PROPERTY PUBLIC StopRequested : BOOL
GET
StopRequested := CycleStopReq;
END_GET
SET // PUBLIC
CycleStopReq := StopRequested;
END_SET
END_PROPERTY

END_FUNCTION_BLOCK

// ---- POUs/PrimeMover.TcPOU
FUNCTION_BLOCK PUBLIC PrimeMover
VAR_IN_OUT
	
END_VAR
VAR_INPUT
END_VAR
VAR_OUTPUT
END_VAR
VAR
	bInitialize : BOOL := TRUE;
	State			:	ePrimeMoverState; 
	NextState		:	ePrimeMoverState;	
	ResetCmdStatus 	:	eMM_ResetCmdStatus;
	StartupCmdStatus:	eMM_StartupCmdStatus;
	HLCStatus		:	eMM_HLCStatus;
	
	// CycleControl will send a Trigger
	Trigger: BOOL := FALSE;
	// Temporary loop variable
	COUNTER: UINT := 1;
	VehicleInitMoveTimer : TON;
	bAllVehStopped :BOOL := TRUE;
	StateTimer :TON;
	WaitAfterESTOPTimer : TON;
	SuspendAfterESTOPTimer: TON;
	bFirst : BOOL := TRUE;
END_VAR

IF (bInitialize) THEN
	bInitialize := FALSE;
	// to add all initialization code here
END_IF


CASE State OF

ePrimeMoverState.eMMUnknown:
    Status.PrimeMoverStatusMsg := 'MM: Unknown, Press Start';
	GVL_IO.MM_YEnableMagneMotion := FALSE;
    IF (GVL_IO.MC_XStartPB AND GVL_IO.MC_XAirPressureOK AND GVL_IO.MC_NotEStopped) THEN // wait for start button when powered up or PLC program restarted
		NextState := ePrimeMoverState.eMMConnect;	   
	END_IF

	StateTimer(IN:=TRUE, PT:= T#9.3S); // give a message out every 10 seconds
	IF (StateTimer.Q) THEN
		Logging.fbEventMsg.SendEventMsg(MsgClass := TCEVENTCLASS_STATEINFO, EventID:= Logging.ID_MM_Unknown, SourceID:= Logging.SrcMMPOU);
		StateTimer(IN:=FALSE);
	END_IF


ePrimeMoverState.eMMConnect:
Status.PrimeMoverStatusMsg := 'MM: Socket Connecting';	
IF (Stations.fbMMClient.eState = eSOCKET_CONNECTED) THEN
		Stations.fbMMSendMsg.M_CmdHLCStatus();
		NextState := ePrimeMoverState.eMMCheckStatus;
	END_IF

ePrimeMoverState.eMMCheckStatus:
Status.PrimeMoverStatusMsg := 'MM: Checking HLC Status';
	IF (HLCStatus = eMM_HLCStatus.eHLC_STATE_OPERATIONAL) THEN
		NextState := ePrimeMoverState.eMMSendResetCmd;		
	END_IF	

ePrimeMoverState.eMMSendResetCmd:
Status.PrimeMoverStatusMsg := 'MM: Reseting Path';
	Stations.fbMMSendMsg.M_CmdResetPath();
	ResetCmdStatus := eMM_ResetCmdStatus.eMM_ResetCmdSent;
	NextState := ePrimeMoverState.eMMWaitAccceptResetCmd;

ePrimeMoverState.eMMWaitAccceptResetCmd:
Status.PrimeMoverStatusMsg := 'MM: Waiting Reset Path ACK';
	IF (ResetCmdStatus = eMM_ResetCmdStatus.eMM_ResetCmdAck) THEN
		NextState := ePrimeMoverState.eMMWaitCmplResetCmd;			
	END_IF	

ePrimeMoverState.eMMWaitCmplResetCmd:
Status.PrimeMoverStatusMsg := 'MM: Waiting Reset Cmpl';
IF (ResetCmdStatus = eMM_ResetCmdStatus.eMM_ResetCmdComplete) THEN
		NextState := ePrimeMoverState.eMMSendStartupCmd;			
	END_IF

ePrimeMoverState.eMMSendStartupCmd:
Status.PrimeMoverStatusMsg := 'MM: Starting Up Path';
	Stations.fbMMSendMsg.M_CmdStartupPath();
	StartupCmdStatus := eMM_StartupCmdStatus.eMM_StartupCmdSent;
	NextState := ePrimeMoverState.eMMWaitAcceptStartupCmd;	

ePrimeMoverState.eMMWaitAcceptStartupCmd:
Status.PrimeMoverStatusMsg := 'MM: Waiting Startup ACK';
	IF (StartupCmdStatus = eMM_StartupCmdStatus.eMM_StartupCmdAck) THEN
		NextState := ePrimeMoverState.eMMWaitCmplStartupCmd;			
	END_IF		

ePrimeMoverState.eMMWaitCmplStartupCmd:
Status.PrimeMoverStatusMsg := 'MM: Waiting Startup CMPL';
	IF (StartupCmdStatus = eMM_StartupCmdStatus.eMM_StartupCmdComplete) THEN
		NextState := ePrimeMoverState.eMMWaitCycleControlTrigger;
	END_IF
	
ePrimeMoverState.eMMWaitCycleControlTrigger:
Status.PrimeMoverStatusMsg := 'MM: Waiting Till Safe to Index';
	IF (Trigger) THEN              //Trigger is Sent By Cycle Controller
			//NextState := ePrimeMoverState.eMMSendAllVehiclesToInitPosCmd;     
		GVL_IO.MM_YEnableMagneMotion := TRUE;
		NextState := ePrimeMoverState.eMMReadyAutoRun;     
        Trigger := FALSE;      	
	END_IF

ePrimeMoverState.eMMSendAllVehiclesToInitPosCmd:
   Trigger := FALSE;	
   FOR COUNTER := 1 TO MM_CONST.MAX_VEHICLES BY 1 DO
		Stations.fbMMSendMsg.M_CmdVehToPos(VehicleID:= COUNTER, Flags :=1, Pos := MM_CONST.GOOD_UNLOAD_POS -((COUNTER-1)* (MM_CONST.Vehicle_Length+MM_CONST.MinGapInterVehStationary)/1000), Acc := 2.0, Vel := 2.0);
		NextState := ePrimeMoverState.eMMWaitCmplAllVehiclesAtInitPos;
	END_FOR
		
ePrimeMoverState.eMMWaitCmplAllVehiclesAtInitPos:
	VehicleInitMoveTimer(IN:=TRUE,PT:=T#3S);
	IF (VehicleInitMoveTimer.Q) THEN
		bAllVehStopped := TRUE;			
		FOR COUNTER := 1 TO MM_CONST.MAX_VEHICLES BY 1 DO
			Stations.fbVehicleManager[COUNTER].VehIdle := TRUE;	
			IF (STATUS.MMVehiclesStatus[COUNTER].Velocity > 0.1) THEN //maybe get vehicle stopped by reading flags instead
				  bAllVehStopped :=FALSE;
				  Stations.fbVehicleManager[COUNTER].VehIdle := FALSE; // this additional variable helps for debug
			END_IF
		END_FOR
		IF (bAllVehStopped) THEN
			NextState := ePrimeMoverState.eMMReadyAutoRun;
			VehicleInitMoveTimer(IN:=FALSE);
		END_IF	
	END_IF 

ePrimeMoverState.eMMReadyAutoRun:
//to do handle all exceptions here 
// according to pg. 53 of 210 of MM TCP/IP manual
// When Host Controller wants to issue E-STOP, then first let all the motion come to a stop
// Then issue a Suspend Movement
// Then remove bus power

//To recover from E-STOP
// Enable Bus Power, wait
// Then issue Resume Movement...
Status.PrimeMoverStatusMsg := 'MM: Auto Run';
	IF (GVL_IO.MachineEStopped OR NOT GVL_IO.MC_XAirPressureOK) THEN 
	   SuspendAfterESTOPTimer(IN:=TRUE, PT:= T#2.5S);
	   IF (SuspendAfterESTOPTimer.Q) THEN
		   NextState := ePrimeMoverState.eMMSuspendMovement;
		   SuspendAfterESTOPTimer(IN:=FALSE);
       END_IF		
	ELSE
		SuspendAfterESTOPTimer(IN:=FALSE);
	END_IF

IF (Stations.fbMMMonitor.IsMMJammed) THEN 
	Status.PrimeMoverStatusMsg := 'MM: Jammed';
END_IF

ePrimeMoverState.eMMSuspendMovement:
	IF (bFirst) THEN 
		//Stations.fbMMSendMsg.M_CmdSuspendMov();  //Suspend command is causing more problems as it rejects commands from vehicles for movement
	END_IF
	SuspendAfterESTOPTimer(IN:=TRUE,PT:=T#5S);
	IF (SuspendAfterESTOPTimer.Q) THEN
		NextState := ePrimeMoverState.eMMESTOP;		
		SuspendAfterESTOPTimer(IN:=FALSE);
		WaitAfterESTOPTimer(IN:=FALSE);
	END_IF

ePrimeMoverState.eMMESTOP:
Status.PrimeMoverStatusMsg := 'MM: E-STOPPED';
	GVL_IO.MM_YEnableMagneMotion := FALSE;
   IF (Stations.fbCycleControl.AllowPrimeMoverEnable) THEN // wait for cycle control to tell us we are ready to move
		WaitAfterESTOPTimer(IN:=TRUE, PT:=T#5S);
		GVL_IO.MM_YEnableMagneMotion := TRUE; // Enable Magnemotion D.C. Bus and let all the vehicles move
		IF (WaitAfterESTOPTimer.Q) THEN
			//Stations.fbMMSendMsg.M_CmdResumeMov(); // let all the vehicles move
			WaitAfterESTOPTimer(IN:=FALSE);
			NextState := ePrimeMoverState.eMMReadyAutoRun;
		END_IF
       	   
	END_IF

ePrimeMoverState.eMMResumeMovement:

ePrimeMoverState.eMMError:
// to do handle all exceptions here

END_CASE

IF (State <> NextState) THEN
	bFirst := TRUE;
	StateTimer(IN:=FALSE);
ELSE
	bFirst := FALSE;
END_IF

State := NextState;

AssignStationStatusForHMI();

PROPERTY PUBLIC StartupCmdState : eMM_StartupCmdStatus
SET
StartupCmdStatus := StartupCmdState;
END_SET
END_PROPERTY

PROPERTY PUBLIC WaitingForHomingTrigger : BOOL
GET
WaitingForHomingTrigger := (StartupCmdStatus = eMM_StartupCmdStatus.eMM_StartupCmdComplete) AND (State = ePrimeMoverState.eMMWaitCycleControlTrigger);
END_GET
END_PROPERTY

METHOD PUBLIC ResetPrimeMoverAndPurge : BOOL
VAR_INPUT
END_VAR
State := ePrimeMoverState.eMMUnknown;
NextState := ePrimeMoverState.eMMUnknown;
END_METHOD

PROPERTY PUBLIC ResetCmdState : eMM_ResetCmdStatus
SET
ResetCmdStatus := ResetCmdState;
END_SET
END_PROPERTY

METHOD PUBLIC AssignStationStatusForHMI : BOOL
VAR_INPUT
END_VAR
Status.StationsState[MM_CONST.PRIME_MOVER_HMI_STATE] := State;
CASE State OF 
	ePrimeMoverState.eMMUnknown,ePrimeMoverState.eMMError:
	Status.StationStauts[MM_CONST.PRIME_MOVER_HMI_STATE] := OverallStationStatus.eError;
	
    ePrimeMoverState.eMMConnect,
	ePrimeMoverState.eMMCheckStatus,
	ePrimeMoverState.eMMSendResetCmd,
	ePrimeMoverState.eMMWaitAccceptResetCmd,
	ePrimeMoverState.eMMWaitCmplResetCmd,
	ePrimeMoverState.eMMSendStartupCmd,
	ePrimeMoverState.eMMWaitAcceptStartupCmd,
	ePrimeMoverState.eMMWaitCmplStartupCmd:
		Status.StationStauts[MM_CONST.PRIME_MOVER_HMI_STATE] := OverallStationStatus.eHoming;
	
	ePrimeMoverState.eMMWaitCycleControlTrigger:
        Status.StationStauts[MM_CONST.PRIME_MOVER_HMI_STATE] := OverallStationStatus.eWarning;
		
	ePrimeMoverState.eMMSendAllVehiclesToInitPosCmd,
	ePrimeMoverState.eMMWaitCmplAllVehiclesAtInitPos,	
    ePrimeMoverState.eMMReadyAutoRun:
	    IF (Stations.fbCycleControl.AllowPrimeMoverEnable) THEN
        	Status.StationStauts[MM_CONST.PRIME_MOVER_HMI_STATE] := OverallStationStatus.eRunning;
		ELSE 
			Status.StationStauts[MM_CONST.PRIME_MOVER_HMI_STATE] := OverallStationStatus.eCycleStop;
		END_IF
		
		IF (Stations.fbMMMonitor.IsMMJammed) THEN 
	        Status.StationStauts[MM_CONST.PRIME_MOVER_HMI_STATE] := OverallStationStatus.eError;
        END_IF
	    
		
	ELSE;	
END_CASE
END_METHOD

PROPERTY PUBLIC HLCState : eMM_HLCStatus
SET
HLCStatus := HLCState;
END_SET
END_PROPERTY

PROPERTY PUBLIC Ready : BOOL
GET
Ready := (State = ePrimeMoverState.eMMReadyAutoRun);
END_GET
END_PROPERTY

PROPERTY PUBLIC TriggerAction : BOOL
SET
Trigger := TriggerAction;
END_SET
END_PROPERTY

END_FUNCTION_BLOCK

// ---- POUs/StationManager.TcPOU
FUNCTION_BLOCK PUBLIC StationManager
VAR_INPUT
END_VAR
VAR_OUTPUT
END_VAR
VAR
END_VAR

;

METHOD PUBLIC NotifyStationNewVehArrival : BOOL
VAR_INPUT
	Pos 			:	REAL;
	StationIndex 	:	BYTE;
	VehicleID		:	BYTE;
END_VAR
CASE StationIndex OF

 
MM_CONST.LOAD_1_STA:
	Stations.fbLoad1Sta.VehicleUnderTest := VehicleID;	
    Stations.fbLoad1Sta.Trigger := TRUE;
		

MM_CONST.LOAD_2_STA:
	Stations.fbLoad2Sta.VehicleUnderTest := VehicleID;		   
    Stations.fbLoad2Sta.Trigger := TRUE;
        			
MM_CONST.LOAD_3_STA:
	Stations.fbLoad3Sta.VehicleUnderTest := VehicleID;	
	Stations.fbLoad3Sta.Trigger := TRUE;					

MM_CONST.LOAD_4_STA:					
	Stations.fbLoad4Sta.VehicleUnderTest := VehicleID;
	Stations.fbLoad4Sta.Trigger := TRUE;	

MM_CONST.STOP_BEFORE_VISION_STA:
	Stations.fbOB_StopBeforeVisionSta.VehicleUnderTest := VehicleID;
	Stations.fbOB_StopBeforeVisionSta.Trigger := TRUE;

MM_CONST.VISION_STA:
	Stations.fbVisionSta.VehicleUnderTest := VehicleID;
	Stations.fbVisionSta.Trigger := TRUE;

MM_CONST.PISTON_STA:
	Stations.fbPistonSta.VehicleUnderTest := VehicleID;
	Stations.fbPistonSta.Trigger := TRUE;

MM_CONST.CAP_STA:
	Stations.fbCapInsertSta.VehicleUnderTest := VehicleID;
	Stations.fbCapInsertSta.Trigger := TRUE;

MM_CONST.IB_STOP_ROBOT_CLEAR_STA:
	Stations.fbIB_StopRobotSta.VehicleUnderTest := VehicleID;
	Stations.fbIB_StopRobotSta.Trigger := TRUE;

MM_CONST.REJECT_ULOAD_STA:
	Stations.fbRejectSta.VehicleUnderTest := VehicleID;
	Stations.fbRejectSta.Trigger := TRUE;

MM_CONST.GOOD_UL_1_STA:
	Stations.fbGoodULSta_1.VehicleUnderTest := VehicleID;
	Stations.fbGoodULSta_1.Trigger := TRUE;

MM_CONST.GOOD_UL_2_STA:
	Stations.fbGoodULSta_2.VehicleUnderTest := VehicleID;
	Stations.fbGoodULSta_2.Trigger := TRUE;

MM_CONST.GOOD_UL_3_STA:
	Stations.fbGoodULSta_3.VehicleUnderTest := VehicleID;
	Stations.fbGoodULSta_3.Trigger := TRUE;

MM_CONST.GOOD_UL_4_STA:
	Stations.fbGoodULSta_4.VehicleUnderTest := VehicleID;
	Stations.fbGoodULSta_4.Trigger := TRUE;

(*	
MM_CONST.GOOD_UNLOAD_STA:
	Stations.fbGoodUnloadSta.VehicleUnderTest := VehicleID;
	Stations.fbGoodUnloadSta.Trigger := TRUE;	
 *)   
MM_CONST.OB_STOP_ROBOT_CLEAR_STA:
	Stations.fbOB_StopRobotSta.VehicleUnderTest := VehicleID;  
    Stations.fbOB_StopRobotSta.Trigger := TRUE;
ELSE ;
	
END_CASE
END_METHOD

END_FUNCTION_BLOCK

// ---- POUs/VehicleManager.TcPOU
FUNCTION_BLOCK PUBLIC VehicleManager
VAR_INPUT
	VehicleID		: BYTE;
END_VAR
VAR_OUTPUT
END_VAR
VAR
	
    State 			: eMM_VehicleState := eMM_VehicleState.eVehIdle;
	NextState		: eMM_VehicleState := eMM_VehicleState.eVehIdle;
	NextPos			: REAL := MM_CONST.REJECT_ULOAD_POS;
	NextVel			: REAL := 2.0;
	NextAcc			: REAL := 2.0;
	NextStaIndex	: BYTE := MM_CONST.REJECT_ULOAD_STA;
	CurrStaIndex	: BYTE := MM_CONST.REJECT_ULOAD_STA;
	cmdAck			: BOOL := FALSE;
	cmdCmpl			: BOOL := FALSE;
	TriggerMove		: BOOL := FALSE;
END_VAR

CASE State OF 
	eMM_VehicleState.eVehIdle: //Set Next Move Parameters and then trigger move
	IF (TriggerMove) THEN
		NextState := eMM_VehicleState.eVehMoveCmd_Send;
		TriggerMove := FALSE;
	END_IF
		
	eMM_VehicleState.eVehMoveCmd_Send:	
	    Stations.fbMMSendMsg.M_CmdVehToPos(VehicleID:=VehicleID,Flags:=1,Pos:=NextPos,Acc:=NextAcc,Vel:=NextVel);
		cmdAck := FALSE;
		cmdCmpl := FALSE;
		NextState:= eMM_VehicleState.eVehMoveCmd_WaitAccept; 	
	eMM_VehicleState.eVehMoveCmd_WaitAccept:
		IF (cmdAck) THEN                           //handle cases for timed out here
			NextState := eMM_VehicleState.eVehMoveCmd_WaitCompl;	
            cmdAck := FALSE;		
		END_IF		
	eMM_VehicleState.eVehMoveCmd_WaitCompl:
		IF (cmdCmpl) THEN                         // handle cases for timed out here 
			NextState := eMM_VehicleState.eVehMoveCmd_Compl;
            cmdCmpl := FALSE; 		
		END_IF
	
	eMM_VehicleState.eVehMoveCmd_Reject:
	
    eMM_VehicleState.eVehMoveCmd_Compl:
		NextState := eMM_VehicleState.eVehIdle;
		Stations.fbStationManager.NotifyStationNewVehArrival(Pos:= NextPos, StationIndex:= NextStaIndex, VehicleID:= VehicleID);		
		CurrStaIndex := NextStaIndex;
		
	eMM_VehicleState.eVehMoveTimeOut:
	
    eMM_VehicleState.eError:
	ELSE
	;		
END_CASE
State := NextState;

METHOD PUBLIC M_SetNextMoveParams : BOOL
VAR_INPUT
	Pos :REAL;
	Vel :REAL;
	Acc :REAL;
	StationIndex :BYTE;
END_VAR
NextPos := Pos;
NextVel	:= Vel;
NextAcc	:= Acc;
NextStaIndex := StationIndex;
END_METHOD

PROPERTY PUBLIC MoveCmdAccepted : BOOL
SET
cmdAck := MoveCmdAccepted;
END_SET
END_PROPERTY

PROPERTY PUBLIC MoveCmdCmpl : BOOL
SET
cmdCmpl := MoveCmdCmpl;
END_SET
END_PROPERTY

METHOD PUBLIC ResetVehicleManager : BOOL
VAR_INPUT
END_VAR
    State 			 := eMM_VehicleState.eVehIdle;
	NextState		 := eMM_VehicleState.eVehIdle;
	NextPos			 := MM_CONST.REJECT_ULOAD_POS;
	NextVel			 := 2.0;
	NextAcc			 := 2.0;
	NextStaIndex	 := MM_CONST.REJECT_ULOAD_STA;
	CurrStaIndex	 := MM_CONST.REJECT_ULOAD_STA;
	cmdAck			 := FALSE;
	cmdCmpl			 := FALSE;
	TriggerMove		 := FALSE;
END_METHOD

METHOD PUBLIC ResetVehicleManagerState : BOOL
VAR_INPUT
END_VAR
State := eMM_VehicleState.eVehIdle;
NextState := eMM_VehicleState.eVehIdle;
END_METHOD

PROPERTY PUBLIC TriggerVehMov : BOOL
SET
TriggerMove := TriggerVehMov;
END_SET
END_PROPERTY

PROPERTY PUBLIC VehIdle : BOOL
GET
VehIdle := (State=eMM_VehicleState.eVehIdle);
END_GET
SET
State:=eMM_VehicleState.eVehIdle;
END_SET
END_PROPERTY

END_FUNCTION_BLOCK

// ---- POUs/RoutePlanner.TcPOU
FUNCTION_BLOCK PUBLIC RoutePlanner
VAR_INPUT
END_VAR
VAR_OUTPUT
END_VAR
VAR
	RejecLoadPosChoice			:       UINT :=5;
	RejectNextStationLocation	:		REAL;
	RejectNextStationIndex		:		BYTE;
	
	GoodULPosChoice				:       UINT :=5;
	GoodULNextStationLocation	:		REAL;
	GoodULNextStationIndex		:		BYTE;
	GoodFullCount : UINT := 0;
	PremiumFullCount : UINT := 0;
	GoodUL_1_NextStationFlag : BYTE := 5; // Next Station is defaulted to 5 ( reject)
	GoodUL_2_NextStationFlag : BYTE := 5; // Next Station is defaulted to 5 ( reject)
	GoodUL_3_NextStationFlag : BYTE := 5; // Next Station is defaulted to 5 ( reject)
	GoodUL_4_NextStationFlag : BYTE := 5; // Next Station is defaulted to 5 ( reject)
END_VAR

;

METHOD PUBLIC M_ExitCapInsertSta : BOOL
VAR_INPUT
	VehicleID		:	BYTE;
END_VAR
IF (PartsData.Status[VehicleID].OverallStatus <> ePartStatus.eReject AND 
    PartsData.Status[VehicleID].OverallStatus <> ePartStatus.eEmpty ) THEN  // we have a good part
   IF (LotsData.Lot.GoodUnloadEnabled) THEN // Good Unload is Enabled
		MoveToGoodUnload(VehicleID);
	ELSE // just go to reject
		MoveToReject(VehicleID);		
	END_IF		
ELSE  // we have a reject	
	MoveToReject(VehicleID);			
END_IF



(*

IF (PartsData.Status[VehicleID].OverallStatus = ePartStatus.eCapInserted) THEN
	Stations.fbVehicleManager[VehicleID].M_SetNextMoveParams(Pos:= MM_CONST.GOOD_UNLOAD_POS, Vel := 2.0, Acc := 2.0, StationIndex := MM_CONST.GOOD_UNLOAD_STA );
	Stations.fbVehicleManager[VehicleID].TriggerVehMov := TRUE;
ELSE 
	Stations.fbVehicleManager[VehicleID].M_SetNextMoveParams(Pos:= MM_CONST.REJECT_ULOAD_POS, Vel := 2.0, Acc := 2.0, StationIndex := MM_CONST.REJECT_ULOAD_STA );
 	Stations.fbVehicleManager[VehicleID].TriggerVehMov := TRUE;		
END_IF
*)

(*
Stations.fbVehicleManager[VehicleID].M_SetNextMoveParams(Pos:= MM_CONST.REJECT_ULOAD_POS, Vel := 2.0, Acc := 2.0, StationIndex := MM_CONST.REJECT_ULOAD_STA );
Stations.fbVehicleManager[VehicleID].TriggerVehMov := TRUE;
*)
END_METHOD

METHOD PUBLIC M_ExitGoodUnload : BOOL
VAR_INPUT
	VehicleID		:	BYTE;
END_VAR
MoveToReject(VehicleID);
END_METHOD

METHOD PUBLIC M_ExitGoodUnload_1 : BOOL
VAR_INPUT
	VehicleID		:	BYTE;
END_VAR
CASE GoodUL_1_NextStationFlag OF
	
    2:	
		MoveToGoodUnload_2(VehicleID);	
	
    3:
		MoveToGoodUnload_3(VehicleID);	
	
    4:
		MoveToGoodUnload_4(VehicleID);	
 
ELSE
		 MoveToReject(VehicleID);
	
END_CASE;
END_METHOD

METHOD PUBLIC M_ExitGoodUnload_2 : BOOL
VAR_INPUT
	VehicleID		:	BYTE;
END_VAR
CASE GoodUL_2_NextStationFlag OF
	
	
    3:
		MoveToGoodUnload_3(VehicleID);	
	
    4:
		MoveToGoodUnload_4(VehicleID);	
 
ELSE
		 MoveToReject(VehicleID);
	
END_CASE;
END_METHOD

METHOD PUBLIC M_ExitGoodUnload_3 : BOOL
VAR_INPUT
	VehicleID		:	BYTE;
END_VAR
CASE GoodUL_3_NextStationFlag OF
	

    4:
		MoveToGoodUnload_4(VehicleID);	
 
ELSE
		 MoveToReject(VehicleID);
	
END_CASE;
END_METHOD

METHOD PUBLIC M_ExitGoodUnload_4 : BOOL
VAR_INPUT
	VehicleID		:	BYTE;
END_VAR
MoveToReject(VehicleID);
END_METHOD

METHOD PUBLIC M_ExitIB_StopRobotClear : BOOL
VAR_INPUT
	VehicleID		:	BYTE;
END_VAR
IF (PartsData.Status[VehicleID].OverallStatus <> ePartStatus.eReject AND 
    PartsData.Status[VehicleID].OverallStatus <> ePartStatus.eEmpty ) THEN  // we have a good part
   IF (LotsData.Lot.CapInsertEnabled) THEN // Cap Is Enabled
		MoveToCap(VehicleID);
	ELSIF (LotsData.Lot.GoodUnloadEnabled) THEN // Good Unload is Enabled
		MoveToGoodUnload(VehicleID);
	ELSE // just go to reject
		MoveToReject(VehicleID);		
	END_IF		
ELSE  // we have a reject	
	MoveToReject(VehicleID);			
END_IF
END_METHOD

METHOD PUBLIC M_ExitLoad1Sta : BOOL
VAR_INPUT
	VehicleID		:	BYTE;
END_VAR
MoveToVision(VehicleID);
//MoveToStopBeforeVision(VehicleID);
END_METHOD

METHOD PUBLIC M_ExitLoad2Sta : BOOL
VAR_INPUT
	VehicleID		:	BYTE;
END_VAR
MoveToVision(VehicleID);
//MoveToStopBeforeVision(VehicleID);
END_METHOD

METHOD PUBLIC M_ExitLoad3Sta : BOOL
VAR_INPUT
	VehicleID		:	BYTE;
END_VAR
MoveToVision(VehicleID);
//MoveToStopBeforeVision(VehicleID);
END_METHOD

METHOD PUBLIC M_ExitLoad4Sta : BOOL
VAR_INPUT
	VehicleID		:	BYTE;
END_VAR
MoveToVision(VehicleID);
//MoveToStopBeforeVision(VehicleID);
END_METHOD

METHOD PUBLIC M_ExitPistonInsertSta : BOOL
VAR_INPUT
	VehicleID		:	BYTE;
END_VAR
IF (PartsData.Status[VehicleID].OverallStatus <> ePartStatus.eReject AND 
    PartsData.Status[VehicleID].OverallStatus <> ePartStatus.eEmpty ) THEN  // we have a good part
    IF (Stations.fbLoad1Sta.HoldVehicle_IBStop) THEN //Yushin wants to load 
		MoveToIBStopRobotClear(VehicleID);
	ELSIF (LotsData.Lot.CapInsertEnabled) THEN // Cap Is Enabled
		MoveToCap(VehicleID);
	ELSIF (LotsData.Lot.GoodUnloadEnabled) THEN // Good Unload is Enabled
		MoveToGoodUnload(VehicleID);
	ELSE // just go to reject
		MoveToReject(VehicleID);		
	END_IF		
ELSE  // we have a reject	
	IF (Stations.fbLoad1Sta.HoldVehicle_IBStop) THEN //Yushin wants to load 
		MoveToIBStopRobotClear(VehicleID);
	ELSE  // just go to reject
		MoveToReject(VehicleID);			
	END_IF
END_IF

(*
IF (Stations.fbLoad1Sta.HoldVehicle_IBStop) THEN //Yushin wants to load 
	Stations.fbVehicleManager[VehicleID].M_SetNextMoveParams(Pos:= MM_CONST.IB_STOP_ROBOT_CLEAR_POS, Vel := 2.0, Acc := 2.0, StationIndex := MM_CONST.IB_STOP_ROBOT_CLEAR_STA );
	Stations.fbVehicleManager[VehicleID].TriggerVehMov := TRUE;
ELSE // move straight to the cap station or reject based on part status
    IF (PartsData.Status[VehicleID].OverallStatus = ePartStatus.ePistonInserted) THEN
		 Stations.fbVehicleManager[VehicleID].M_SetNextMoveParams(Pos:= MM_CONST.CAP_POS, Vel := 2.0, Acc := 2.0, StationIndex := MM_CONST.CAP_STA );
		 Stations.fbVehicleManager[VehicleID].TriggerVehMov := TRUE;
	ELSE 
		Stations.fbVehicleManager[VehicleID].M_SetNextMoveParams(Pos:= MM_CONST.REJECT_ULOAD_POS, Vel := 2.0, Acc := 2.0, StationIndex := MM_CONST.REJECT_ULOAD_STA );
 		Stations.fbVehicleManager[VehicleID].TriggerVehMov := TRUE;
	END_IF
   
END_IF



//Stations.fbVehicleManager[VehicleID].M_SetNextMoveParams(Pos:= MM_CONST.CAP_POS, Vel := 2.0, Acc := 2.0, StationIndex := MM_CONST.CAP_STA );
//Stations.fbVehicleManager[VehicleID].TriggerVehMov := TRUE;


// Stations.fbVehicleManager[VehicleID].M_SetNextMoveParams(Pos:= MM_CONST.REJECT_ULOAD_POS, Vel := 2.0, Acc := 2.0, StationIndex := MM_CONST.REJECT_ULOAD_STA );
 // Stations.fbVehicleManager[VehicleID].TriggerVehMov := TRUE;


(*

	Stations.fbVehicleManager[VehicleID].M_SetNextMoveParams(Pos:= MM_CONST.PISTON_POS, Vel := 2.0, Acc := 2.0, StationIndex := MM_CONST.PISTON_STA );
	Stations.fbVehicleManager[VehicleID].TriggerVehMov := TRUE;
	*)

(*


IF (Stations.fbLoad1Sta.HoldVehicle_IBStop) THEN //Yushin wants to load 
	Stations.fbVehicleManager[VehicleID].M_SetNextMoveParams(Pos:= MM_CONST.IB_STOP_ROBOT_CLEAR_POS, Vel := 2.0, Acc := 2.0, StationIndex := MM_CONST.IB_STOP_ROBOT_CLEAR_STA );
	Stations.fbVehicleManager[VehicleID].TriggerVehMov := TRUE;
ELSE // move straight to the cap station
	// NEED TO REMOVE THIS AFTER DEBUG ON 3/19/2017... WE ARE BYPASSING CAP STATION FOR NOW 
    //Stations.fbVehicleManager[VehicleID].M_SetNextMoveParams(Pos:= MM_CONST.CAP_POS, Vel := 2.0, Acc := 2.0, StationIndex := MM_CONST.CAP_STA );
	//Stations.fbVehicleManager[VehicleID].TriggerVehMov := TRUE;
	
	Stations.fbVehicleManager[VehicleID].M_SetNextMoveParams(Pos:= MM_CONST.GOOD_UNLOAD_POS, Vel := 2.0, Acc := 2.0, StationIndex := MM_CONST.GOOD_UNLOAD_STA );
	Stations.fbVehicleManager[VehicleID].TriggerVehMov := TRUE;
			
END_IF

*)
*)
END_METHOD

METHOD PUBLIC M_ExitRejectUnload : BOOL
VAR_INPUT	
	VehicleID		:	BYTE;
END_VAR
RejecLoadPosChoice := RejecLoadPosChoice -1; //we initialize with this variable as 5;
IF (RejecLoadPosChoice<=0 OR RejecLoadPosChoice>=4 ) THEN 
	RejecLoadPosChoice := 4;
END_IF
CASE RejecLoadPosChoice OF
				4: 
					RejectNextStationLocation := MM_CONST.OB_STOP_ROBOT_CLEAR_POS;
					RejectNextStationIndex	:= MM_CONST.OB_STOP_ROBOT_CLEAR_STA;
				3:
					RejectNextStationLocation := MM_CONST.LOAD_3_POS;
					RejectNextStationIndex	:= MM_CONST.LOAD_3_STA;
				2:
					RejectNextStationLocation := MM_CONST.LOAD_2_POS;
					RejectNextStationIndex	:= MM_CONST.LOAD_2_STA;
				1:
					RejectNextStationLocation := MM_CONST.LOAD_1_POS;
					RejectNextStationIndex	:= MM_CONST.LOAD_1_STA;						
END_CASE				
	
Stations.fbVehicleManager[VehicleID].M_SetNextMoveParams(Pos:= RejectNextStationLocation, Vel := 2.0, Acc := 2.0, StationIndex := RejectNextStationIndex );
Stations.fbVehicleManager[VehicleID].TriggerVehMov := TRUE;
END_METHOD

METHOD PUBLIC M_ExitVisionSta : BOOL
VAR_INPUT
	VehicleID		:	BYTE;
END_VAR
IF (PartsData.Status[VehicleID].OverallStatus <> ePartStatus.eReject AND 
    PartsData.Status[VehicleID].OverallStatus <> ePartStatus.eEmpty ) THEN  // we have a good part
    IF (LotsData.Lot.PistonInsertEnabled) THEN //Piston is enabled
		MoveToPiston(VehicleID);
	ELSIF (Stations.fbLoad1Sta.HoldVehicle_IBStop) THEN //Yushin wants to load 
		MoveToIBStopRobotClear(VehicleID);
	ELSIF (LotsData.Lot.CapInsertEnabled) THEN // If Cap Is Enabled
		MoveToCap(VehicleID);		
	ELSIF (LotsData.Lot.GoodUnloadEnabled) THEN // If Good Unload is Enabled
		MoveToGoodUnload(VehicleID);
	ELSE // just go to reject
		MoveToReject(VehicleID);	
	END_IF		
ELSE  // we have a reject	
	IF (Stations.fbLoad1Sta.HoldVehicle_IBStop) THEN //Yushin wants to load 
		MoveToIBStopRobotClear(VehicleID);
	ELSE  // just go to reject
		MoveToReject(VehicleID);		
	END_IF
END_IF
END_METHOD

METHOD PUBLIC M_NotifyVehStaCmpl : BOOL
VAR_INPUT
	StationIndex 	:	BYTE;
	VehicleID		:	BYTE;
END_VAR
CASE StationIndex OF

		
	MM_CONST.LOAD_1_STA:
        M_ExitLoad1Sta(VehicleID := VehicleID);

    MM_CONST.LOAD_2_STA:
		M_ExitLoad2Sta(VehicleID := VehicleID);

    MM_CONST.LOAD_3_STA:
		M_ExitLoad3Sta(VehicleID := VehicleID);			

    MM_CONST.LOAD_4_STA:					
       M_ExitLoad4Sta(VehicleID := VehicleID);

    MM_CONST.STOP_BEFORE_VISION_STA:
		M_OBExit_StopBeforeVision(VehicleID := VehicleID);

    MM_CONST.VISION_STA:
		M_ExitVisionSta(VehicleID := VehicleID);

    MM_CONST.PISTON_STA:		
		M_ExitPistonInsertSta(VehicleID := VehicleID);

	MM_CONST.IB_STOP_ROBOT_CLEAR_STA:
		M_ExitIB_StopRobotClear(VehicleID := VehicleID);
    
    MM_CONST.CAP_STA:
		M_ExitCapInsertSta(VehicleID := VehicleID);
   
    MM_CONST.GOOD_UNLOAD_STA:	
	   M_ExitGoodUnload(VehicleID:=VehicleID);  

    MM_CONST.GOOD_UL_1_STA:
		M_ExitGoodUnload_1(VehicleID:=VehicleID); 
	
	MM_CONST.GOOD_UL_2_STA:
		M_ExitGoodUnload_2(VehicleID:=VehicleID); 
		
	MM_CONST.GOOD_UL_3_STA:
		M_ExitGoodUnload_3(VehicleID:=VehicleID); 
	
	MM_CONST.GOOD_UL_4_STA:	
		M_ExitGoodUnload_4(VehicleID:=VehicleID); 
  

    MM_CONST.REJECT_ULOAD_STA:		
		M_ExitRejectUnload(VehicleID:= VehicleID);
	
	MM_CONST.OB_STOP_ROBOT_CLEAR_STA:
		M_OBExitOB_StopBeforeRobotClear(VehicleID := VehicleID);

ELSE; 
END_CASE
END_METHOD

METHOD PUBLIC M_OBExit_StopBeforeVision : BOOL
VAR_INPUT
	VehicleID		:	BYTE;
END_VAR
IF (PartsData.Status[VehicleID].OverallStatus = ePartStatus.eEmpty) THEN
  MoveToReject(VehicleID);
ELSE	
    MoveToVision(VehicleID);
END_IF
END_METHOD

METHOD PUBLIC M_OBExitOB_StopBeforeRobotClear : BOOL
VAR_INPUT
	VehicleID: BYTE;
END_VAR
MoveToLoadPos4(VehicleID);
END_METHOD

METHOD PUBLIC MoveToCap : BOOL
VAR_INPUT
	VehicleID		:	BYTE;
END_VAR
Stations.fbVehicleManager[VehicleID].M_SetNextMoveParams(Pos:= MM_CONST.CAP_POS, Vel := 2.0, Acc := 2.0, StationIndex := MM_CONST.CAP_STA );
Stations.fbVehicleManager[VehicleID].TriggerVehMov := TRUE;
END_METHOD

METHOD PUBLIC MoveToGoodUnload : BOOL
VAR_INPUT
	VehicleID		:	BYTE;
END_VAR
// If for some reason a reject parts comes here, send it to reject station
	IF (PartsData.Status[VehicleID].OverallStatus = ePartStatus.eReject) THEN
		MoveToReject(VehicleID);
		RETURN; 
	END_IF	

// If the Auto-Bagger is not enabled, then we distribute the pallets to all 2 UL stations 

IF (NOT LotsData.Lot.AutoBaggerEnabled) THEN
	IF (PartsData.Status[VehicleID].Premium) THEN
		MoveToGoodUnload_2(VehicleID);
	ELSIF (PartsData.Status[VehicleID].Good) THEN
        MoveToGoodUnload_3(VehicleID);
	ELSE
		MoveToReject(VehicleID);
	END_IF
	
		// Reset all Chute Part Counters 
	Config.PremiumCount1 := 0;
	Config.PremiumCount2 := 0;
	Config.GoodCount1 := 0;
	Config.GoodCount2 := 0;
	GoodFullCount := 0;
    PremiumFullCount := 0;
	
	// Exit from this routine
	RETURN;
END_IF
 
// If Auto-bagger is enabled  
// Chute choice is relegated at the individual station
IF (PartsData.Status[VehicleID].Premium) THEN
	MoveToGoodUnload_1(VehicleID);	
ELSIF (PartsData.Status[VehicleID].Good) THEN
	MoveToGoodUnload_3(VehicleID);
ELSE
	MoveToReject(VehicleID);
END_IF

(*
IF (PartsData.Status[VehicleID].Premium) THEN
	    // First preference is to fill Chute closest to Reject Station. 
		IF((Config.PremiumCount1 < LotsData.Lot.QuantityInBag) AND ((Config.PremiumCount2 < (LotsData.Lot.QuantityInBag-10)) OR (Config.PremiumCount2 = LotsData.Lot.QuantityInBag))) THEN
			MoveToGoodUnload_1(VehicleID);			
			PremiumFullCount := 0;
		ELSIF (Config.PremiumCount2 < LotsData.Lot.QuantityInBag) THEN
			MoveToGoodUnload_2(VehicleID);			
			PremiumFullCount := 0;
		ELSE  // demote the status of the parts to Good
			PartsData.Status[VehicleID].Premium := FALSE;
			PartsData.Status[VehicleID].Good := TRUE;
			PremiumFullCount := PremiumFullCount + 1;
		END_IF
	END_IF

// If the Parts are Good 	
	IF (PartsData.Status[VehicleID].Good) THEN   
		//First preference is to fill the Chute downstream closer to reject/premium 
		IF ((Config.GoodCount1 < LotsData.Lot.QuantityInBag) AND ((Config.GoodCount2 < (LotsData.Lot.QuantityInBag-10)) OR (Config.GoodCount2 = LotsData.Lot.QuantityInBag))) THEN
			MoveToGoodUnload_3(VehicleID);	
			GoodFullCount := 0;
		ELSIF (Config.GoodCount2 < LotsData.Lot.QuantityInBag) THEN
			MoveToGoodUnload_4(VehicleID);	
			GoodFullCount := 0;
		ELSE
			PartsData.Status[VehicleID].Premium := FALSE;
			PartsData.Status[VehicleID].Good := FALSE;
			PartsData.Status[VehicleID].OverallStatus := ePartStatus.eReject;
			PartsData.Status[VehicleID].GoodUnload := FALSE;
			GoodFullCount := GoodFullCount + 1;
		END_IF	
	END_IF
    	
	IF (PartsData.Status[VehicleID].OverallStatus = ePartStatus.eReject) THEN
		MoveToReject(VehicleID);
	END_IF	
	
	IF (GoodFullCount >= 5 OR PremiumFullCount >= 5) THEN
		Stations.fbCycleControl.StopRequested := TRUE;
		Status.AutoBaggerStatusMsg := 'AutoBagger: No drop location available. Clear Chutes';
	END_IF	
	
*)
END_METHOD

METHOD PUBLIC MoveToGoodUnload_1 : BOOL
VAR_INPUT
	VehicleID		:	BYTE;
END_VAR
Stations.fbVehicleManager[VehicleID].M_SetNextMoveParams(Pos:= MM_CONST.GOOD_UL_1_POS, Vel := 2.0, Acc := 2.0, StationIndex := MM_CONST.GOOD_UL_1_STA );
Stations.fbVehicleManager[VehicleID].TriggerVehMov := TRUE;
END_METHOD

METHOD PUBLIC MoveToGoodUnload_2 : BOOL
VAR_INPUT
	VehicleID		:	BYTE;
END_VAR
Stations.fbVehicleManager[VehicleID].M_SetNextMoveParams(Pos:= MM_CONST.GOOD_UL_2_POS, Vel := 2.0, Acc := 2.0, StationIndex := MM_CONST.GOOD_UL_2_STA );
Stations.fbVehicleManager[VehicleID].TriggerVehMov := TRUE;
END_METHOD

METHOD PUBLIC MoveToGoodUnload_3 : BOOL
VAR_INPUT
	VehicleID		:	BYTE;
END_VAR
Stations.fbVehicleManager[VehicleID].M_SetNextMoveParams(Pos:= MM_CONST.GOOD_UL_3_POS, Vel := 2.0, Acc := 2.0, StationIndex := MM_CONST.GOOD_UL_3_STA );
Stations.fbVehicleManager[VehicleID].TriggerVehMov := TRUE;
END_METHOD

METHOD PUBLIC MoveToGoodUnload_4 : BOOL
VAR_INPUT
	VehicleID		:	BYTE;
END_VAR
Stations.fbVehicleManager[VehicleID].M_SetNextMoveParams(Pos:= MM_CONST.GOOD_UL_4_POS, Vel := 2.0, Acc := 2.0, StationIndex := MM_CONST.GOOD_UL_4_STA );
Stations.fbVehicleManager[VehicleID].TriggerVehMov := TRUE;
END_METHOD

METHOD PUBLIC MoveToIBStopRobotClear : BOOL
VAR_INPUT
	VehicleID		:	BYTE;
END_VAR
Stations.fbVehicleManager[VehicleID].M_SetNextMoveParams(Pos:= MM_CONST.IB_STOP_ROBOT_CLEAR_POS, Vel := 2.0, Acc := 2.0, StationIndex := MM_CONST.IB_STOP_ROBOT_CLEAR_STA );
Stations.fbVehicleManager[VehicleID].TriggerVehMov := TRUE;
END_METHOD

METHOD PUBLIC MoveToLoadPos4 : BOOL
VAR_INPUT
	VehicleID		:	BYTE;
END_VAR
Stations.fbVehicleManager[VehicleID].M_SetNextMoveParams(Pos:= MM_CONST.LOAD_4_POS, Vel := 2.0, Acc := 2.0, StationIndex := MM_CONST.LOAD_4_STA );
Stations.fbVehicleManager[VehicleID].TriggerVehMov := TRUE;
END_METHOD

METHOD PUBLIC MoveToPiston : BOOL
VAR_INPUT
	VehicleID		:	BYTE;
END_VAR
Stations.fbVehicleManager[VehicleID].M_SetNextMoveParams(Pos:= MM_CONST.PISTON_POS, Vel := 2.0, Acc := 2.0, StationIndex := MM_CONST.PISTON_STA );
Stations.fbVehicleManager[VehicleID].TriggerVehMov := TRUE;
END_METHOD

METHOD PUBLIC MoveToReject : BOOL
VAR_INPUT
	VehicleID		:	BYTE;
END_VAR
Stations.fbVehicleManager[VehicleID].M_SetNextMoveParams(Pos:= MM_CONST.REJECT_ULOAD_POS, Vel := 2.0, Acc := 2.0, StationIndex := MM_CONST.REJECT_ULOAD_STA );
Stations.fbVehicleManager[VehicleID].TriggerVehMov := TRUE;
END_METHOD

METHOD PUBLIC MoveToStopBeforeVision : BOOL
VAR_INPUT
	VehicleID		:	BYTE;
END_VAR
Stations.fbVehicleManager[VehicleID].M_SetNextMoveParams(Pos:= MM_CONST.STOP_BEFORE_VISION_POS, Vel := 2.0, Acc := 0.5, StationIndex := MM_CONST.STOP_BEFORE_VISION_STA);
Stations.fbVehicleManager[VehicleID].TriggerVehMov := TRUE;
END_METHOD

METHOD PUBLIC MoveToVision : BOOL
VAR_INPUT
	VehicleID		:	BYTE;
END_VAR
Stations.fbVehicleManager[VehicleID].M_SetNextMoveParams(Pos:= MM_CONST.VISION_POS, Vel := 2.0, Acc := 2.0, StationIndex := MM_CONST.VISION_STA );
Stations.fbVehicleManager[VehicleID].TriggerVehMov := TRUE;
END_METHOD

PROPERTY PUBLIC P_GoodUnload_1_NextStaFlag : BYTE
SET
GoodUL_1_NextStationFlag := P_GoodUnload_1_NextStaFlag;
END_SET
END_PROPERTY

PROPERTY PUBLIC P_GoodUnload_2_NextStaFlag : BYTE
SET
GoodUL_2_NextStationFlag := P_GoodUnload_2_NextStaFlag;
END_SET
END_PROPERTY

PROPERTY PUBLIC P_GoodUnload_3_NextStaFlag : BYTE
SET
GoodUL_3_NextStationFlag := P_GoodUnload_3_NextStaFlag;
END_SET
END_PROPERTY

PROPERTY PUBLIC P_GoodUnload_4_NextStaFlag : BYTE
SET
GoodUL_4_NextStationFlag := P_GoodUnload_4_NextStaFlag;
END_SET
END_PROPERTY

METHOD SetGoodULLoadPosChoiceToInit : BOOL
VAR_INPUT
END_VAR
GoodULPosChoice	:=5;
END_METHOD

METHOD PUBLIC SetRejectLoadPosChoiceToInit : BOOL
VAR_INPUT
END_VAR
RejecLoadPosChoice := 5;
END_METHOD

END_FUNCTION_BLOCK

// ---- POUs/Load1Station.TcPOU
// This Station Interacts with the Load Station Tooling as well as the Yushin Robot. It also signals the Inbound track to hold parts when the Yushin wants to engage 
FUNCTION_BLOCK PUBLIC Load1Station
VAR_INPUT
END_VAR
VAR_OUTPUT
END_VAR
VAR
	xTrigger :BOOL := FALSE; // triggers processing
	State : eLoadSta1State := eLoadSta1State.eUnknown;
	NextState : eLoadSta1State := eLoadSta1State.eUnknown;
	ErrorReturnState : eLoadSta1State := eLoadSta1State.eUnknown;
	bFirst : BOOL := TRUE;
	VUT : BYTE; //VehicleID Under Station
	DwellTimer : TON;
	LoadingComplete : BOOL := FALSE;
	HoldVehicleAtIBStop: BOOL := FALSE;
	StateTimer : TON;
	YushinTimer : TON;
	CycleNumb: INT :=0;
	RowNumber :INT:=0;
	SeedNumber : INT:=13;
END_VAR

IF (GVL_IO.MachineEStopped) THEN 
	State := eLoadSta1State.eUnknown;
	NextState := eLoadSta1State.eUnknown;	
END_IF


CASE State OF

eLoadSta1State.eUnknown:
	IF (GVL_IO.MC_XStartPB AND GVL_IO.MC_XAirPressureOK AND GVL_IO.MC_NotEStopped) THEN // wait for start button when powered up or PLC program restarted
		NextState := eLoadSta1State.eInit;	   
	END_IF	
    IF (GVL_IO.MachineEStopped) THEN
		Status.Load1StatusMsg:= 'Load: E-Stopped. Press Reset';
	ELSIF (NOT GVL_IO.MC_XAirPressureOK) THEN
		Status.Load1StatusMsg:= 'Load: No Air Pressure. Check Air Pressure/Sensor';
	ELSE
		Status.Load1StatusMsg:= 'Load: Reset Ok, Air OK. Press Start Button';			
	END_IF
    
	Status.BurnOffIdle := TRUE;
	
eLoadSta1State.eInit:
	Act_FreePalletHoldDown();
	Act_FreePalletRelease();
	Act_RetractPalletClose();
	ResetDwellTimer();
	NextState := eLoadSta1State.eHoming;	
	
    
	

eLoadSta1State.eHoming:
	Status.Load1StatusMsg:= 'Load: Homing Pallet HoldDown And Release Cylinders';
    IF (IsPalletHoldDownFree() AND IsPalletReleaseFree() AND IsPalletCloseRetracted()) THEN
		Status.BurnOffIdle := FALSE; 
        IF(xTrigger) THEN  //we are recovering from E-STOP or I/O Lock and haven't released prior pallets
		 NextState := eLoadSta1State.eProcessing; 
		ELSE
			NextState := eLoadSta1State.eReady; //wait for all parts to show up 
		END_IF
        
	END_IF
   
   DwellTimer(IN:= TRUE, PT:= T#10S);
   IF (DwellTimer.Q) THEN
	   ResetDwellTimer();
	   ErrorReturnState:= eLoadSta1State.eInit;	   
   	   NextState := eLoadSta1State.eError;	
   END_IF 
	
		

eLoadSta1State.eReady:  //Wait here until part arrives -- this also assumes that Vehicles have arrived at LoadStation 2, 3 and 4.. To Do check and confirm this
	Status.Load1StatusMsg:= 'Load: Waiting all four pallets to arrive';	
    IF (xTrigger) THEN
		NextState := eLoadSta1State.eWaitForYushinPrepareLoad;			
		ResetDwellTimer();
		ResetStateTimer();
	END_IF	
	
eLoadSta1State.eWaitForYushinPrepareLoad:  //here is where the Yushin will signal that are parts ready to be loaded
   IF (NOT IsPalletHoldDownFree()) THEN
       Act_FreePalletHoldDown();
   END_IF
   IF (NOT IsPalletReleaseFree()) THEN
	   Act_FreePalletRelease();
   END_IF
   IF (NOT IsPalletCloseRetracted()) THEN
	   Act_RetractPalletClose();
   END_IF
      
   Status.Load1StatusMsg:= 'Load: Waiting For Yushin';
    IF (GVL_IO.YU_XPrepareToLoad (* OR TRUE*) ) THEN    //debug mode loctite  ///Turnkey shop debug added OR TRUE
	   RowNumber := 0;
       RowNumber.0 := GVL_IO.YU_XLocBit0;
	   RowNumber.1 := GVL_IO.YU_XLocBit1;
	   GVL_IO.YU_YOkToLoad := FALSE;
	   ResetDwellTimer();
	   HoldVehicleAtIBStop:= FALSE;  // don't even do it for row 4
	   //NextState := eLoadSta1State.ePalletHoldDownEngage; 
	   NextState := eLoadSta1State.ePalletReleaseRaise; //new sequence 8/5 
	   IF (GVL_IO.YU_XLocBit1 AND GVL_IO.YU_XLocBit0) THEN //row 4 only
		   //HoldVehicleAtIBStop:= TRUE;
		  // NextState := eLoadSta1State.eWaitForIBTrackClear;		
   	  END_IF
    END_IF 
   StateTimer(IN:=TRUE, PT:= T#90S); // give a message out every 10 seconds
   IF (StateTimer.Q) THEN
	   Status.BurnOffIdle := TRUE;
   END_IF
   
 
eLoadSta1State.eWaitForIBTrackClear: // read the location bits from Yushin in this state and decide what to do with traffic stop
	DwellTimer(IN:=IsInBoundTrackClear(), PT := T#1000MS);
	Act_EngagePalletHoldDown(); //doing actions in parallel to speed things up
	IF (IsPalletHoldDownEngaged()) THEN
		Act_EngagePalletRelease();
	END_IF
	IF (DwellTimer.Q) THEN
		NextState := eLoadSta1State.ePalletHoldDownEngage;
        // NextState := eLoadSta1State.eSignalYushinOKToLoad;
		//NextState := eLoadSta1State.eWaitForYushinToolDown;	
		DwellTimer(IN:=FALSE);
	END_IF

eLoadSta1State.ePalletHoldDownEngage:
	Status.BurnOffIdle := FALSE;
	Act_EngagePalletHoldDown();
	ResetDwellTimer();
	NextState:= eLoadSta1State.ePalletHoldDownEngaged;
		
	
eLoadSta1State.ePalletHoldDownEngaged:
	Status.Load1StatusMsg:= 'Load: Waiting Pallet Hold Down To Be Engaged';
	IF (IsPalletHoldDownEngaged()) THEN
		//NextState := eLoadSta1State.ePalletReleaseRaise;  //new sequence 8/5
		NextState := eLoadSta1State.eSignalYushinOKToLoad;
	END_IF
	
   DwellTimer(IN:= TRUE, PT:= T#10S);
   IF (DwellTimer.Q) THEN
	   ResetDwellTimer();
	   ErrorReturnState:= eLoadSta1State.ePalletHoldDownEngage;	   
   	   NextState := eLoadSta1State.eError;	
   END_IF 
	

eLoadSta1State.ePalletReleaseRaise:
	Act_EngagePalletRelease();
	ResetDwellTimer();
 	NextState := eLoadSta1State.ePalletReleaseRaised;
	
eLoadSta1State.ePalletReleaseRaised:
	Status.Load1StatusMsg:= 'Load: Waiting Pallet Release To Be Engaged';
    IF  (IsPalletReleaseEngaged()) THEN
		//NextState := eLoadSta1State.eSignalYushinOKToLoad;
		NextState := eLoadSta1State.ePalletHoldDownEngage; 
		ResetDwellTimer();
	END_IF
	
   DwellTimer(IN:= TRUE, PT:= T#10S);
   IF (DwellTimer.Q) THEN
	   ResetDwellTimer();
	   ErrorReturnState:= eLoadSta1State.ePalletReleaseRaise;	   
   	   NextState := eLoadSta1State.eError;	
   END_IF 
	
eLoadSta1State.eSignalYushinOKToLoad: 
	GVL_IO.YU_YOkToLoad := TRUE;
	GVL_IO.YU_YAckPartsHeld := FALSE;
	ResetDwellTimer();
	NextState := eLoadSta1State.eWaitForYushinToolDown;
	
    	
eLoadSta1State.eWaitForYushinToolDown:
   Status.Load1StatusMsg:= 'Load: Waiting For Yushin Tool Down';
   ///////
   // Timer section for Turnkey debug in the shop without the robot 
   //////
   //DwellTimer(IN:=TRUE , PT:= T#2S);   //loctite mode 
   
   DwellTimer(IN:=GVL_IO.YU_XToolDown , PT:= T#250MS);   //uncomment this our at Nordson 
   
   IF (DwellTimer.Q) THEN
	   GVL_IO.YU_YOkToLoad := FALSE;
       ResetDwellTimer();   
	   NextState := eLoadSta1State.ePalletCloseExtend;
	   //Act_FreePalletHoldDown();	   
   END_IF
 
eLoadSta1State.ePalletCloseExtend:
 	Act_ExtendPalletClose();
	ResetDwellTimer();
	NextState := eLoadSta1State.ePalletCloseExtended;
	
eLoadSta1State.ePalletCloseExtended:
    IF (IsPalletCloseExtended()) THEN
		ResetDwellTimer();
		NextState := eLoadSta1State.ePalletCloseRetract; 
	END_IF
   
   DwellTimer(IN:= TRUE, PT:= T#10S);
   IF (DwellTimer.Q) THEN
	   ResetDwellTimer();
	   ErrorReturnState:= eLoadSta1State.ePalletCloseExtend;	   
   	   NextState := eLoadSta1State.eError;	
   END_IF 
	
eLoadSta1State.ePalletCloseRetract:
	Act_RetractPalletClose();
	ResetDwellTimer();
	NextState := eLoadSta1State.ePalletCloseRetracted;

eLoadSta1State.ePalletCloseRetracted:
	 IF (IsPalletCloseRetracted()) THEN
		ResetDwellTimer();
		Act_FreePalletRelease();
        NextState := eLoadSta1State.ePalletReleaseLower;	
	END_IF	
	
   DwellTimer(IN:= TRUE, PT:= T#10S);
   IF (DwellTimer.Q) THEN
	   ResetDwellTimer();
	   ErrorReturnState:= eLoadSta1State.ePalletCloseRetract;	   
   	   NextState := eLoadSta1State.eError;	
   END_IF 
   
eLoadSta1State.ePalletReleaseLower:
	Act_FreePalletRelease();
	ResetDwellTimer();
 	NextState := eLoadSta1State.ePalletReleaseLowered;

eLoadSta1State.ePalletReleaseLowered:
     Status.Load1StatusMsg:= 'Load: Waiting Pallet Release To Be Free'; 
	 IF (IsPalletReleaseFree()) THEN
		 ResetDwellTimer();
		 ResetStateTimer();
		 GVL_IO.YU_YAckPartsHeld := TRUE;
		 NextState := eLoadSta1State.eWaitForYushinToolUp;
	 END_IF
	
   DwellTimer(IN:= TRUE, PT:= T#10S);
   IF (DwellTimer.Q) THEN
	   ResetDwellTimer();
	   ErrorReturnState:= eLoadSta1State.ePalletReleaseLower;	   
   	   NextState := eLoadSta1State.eError;	
   END_IF 
    
eLoadSta1State.eWaitForYushinToolUp:
	Status.Load1StatusMsg:= 'Load: Waiting For Yushin Tool Up';
	
	// Timer section only added for Turnkey Debug in the shop
    DwellTimer(IN:=(GVL_IO.YU_XToolUp AND NOT GVL_IO.YU_XToolDown ), PT := T#10MS);   //uncomment this at Nordson
	StateTimer(IN:=TRUE, PT:= T#10S);
	//DwellTimer(IN:=TRUE, PT:= T#100MS);  //only for Turnkey shop
	IF (DwellTimer.Q OR StateTimer.Q) THEN
		HoldVehicleAtIBStop:= FALSE;
		NextState := eLoadSta1State.ePalletHoldDownFree;		
		DwellTimer(IN:=FALSE);
		StateTimer(IN:=FALSE);			
	END_IF
	
eLoadSta1State.ePalletHoldDownFree:
	Act_FreePalletHoldDown();
	ResetDwellTimer();
 	NextState := eLoadSta1State.ePalletHoldDownFreed;

	
eLoadSta1State.ePalletHoldDownFreed:
 	IF (IsPalletHoldDownFree()) THEN 		
		NextState := eLoadSta1State.eProcessing;
		DwellTimer(IN:=FALSE);
		StateTimer(IN:=FALSE);
	END_IF
	
	DwellTimer(IN:= TRUE, PT:= T#10S);
   	IF (DwellTimer.Q) THEN
	   ResetDwellTimer();
	   ErrorReturnState:= eLoadSta1State.ePalletHoldDownFree;	   
   	   NextState := eLoadSta1State.eError;	
   	END_IF 
    
	

eLoadSta1State.eProcessing: // Load Station 1 is directing the other load stations that loading is complete.
	Stations.fbLoad2Sta.SetRowNumber(RowLocationNumber := RowNumber);
    Stations.fbLoad2Sta.LoadComplete := TRUE; 
	Stations.fbLoad3Sta.SetRowNumber(RowLocationNumber := RowNumber);
	Stations.fbLoad3Sta.LoadComplete := TRUE;
	Stations.fbLoad4Sta.SetRowNumber(RowLocationNumber := RowNumber);
	Stations.fbLoad4Sta.LoadComplete := TRUE;
	Stations.fbOB_StopRobotSta.MoveToLoading := TRUE;
    UpdatePartData();	
	NextState := eLoadSta1State.eDepart;

eLoadSta1State.eDepart:
	Stations.fbRoutePlanner.M_NotifyVehStaCmpl(StationIndex:= MM_CONST.LOAD_1_STA, VehicleID := VUT);
	xTrigger := FALSE;
    IF (Stations.fbCycleControl.StopRequested) THEN
        NextState := eLoadSta1State.eStopActive;
    ELSE		
		NextState := eLoadSta1State.eReady;	
	END_IF

eLoadSta1State.eStopActive:
      Status.Load1StatusMsg:= 'Load: Stopped, Press Start';
     IF (NOT Stations.fbCycleControl.StopRequested) THEN
        NextState := eLoadSta1State.eReady;
	END_IF
	
eLoadSta1State.eError:
	IF (GVL_IO.MC_XStartPB) THEN
		NextState := ErrorReturnState;
		ErrorReturnState := eLoadSta1State.eUnknown;
	END_IF

END_CASE

IF (State <> NextState) THEN
	bFirst := TRUE;
	StateTimer(IN:=FALSE);
ELSE
	bFirst := FALSE;
END_IF

State := NextState;
AssignStationStatusForHMI();

ACTION Act_EngagePalletHoldDown:
GVL_IO.LD_YPalletHoldDownExtendHome := FALSE;
GVL_IO.LD_YPalletHoldDownRetractEngage := TRUE;
END_ACTION

ACTION Act_EngagePalletRelease:
GVL_IO.LD_YPalletReleaseExtend := TRUE;
GVL_IO.LD_YPalletReleaseRetract := FALSE;
END_ACTION

ACTION Act_ExtendPalletClose:
GVL_IO.LD_YPalletCloseExtend := TRUE;
GVL_IO.LD_YPalletCloseRetract := FALSE;
END_ACTION

ACTION Act_FreePalletHoldDown:
GVL_IO.LD_YPalletHoldDownExtendHome := TRUE; 
GVL_IO.LD_YPalletHoldDownRetractEngage := FALSE;
END_ACTION

ACTION Act_FreePalletRelease:
GVL_IO.LD_YPalletReleaseExtend := FALSE;
GVL_IO.LD_YPalletReleaseRetract := TRUE;
END_ACTION

ACTION Act_RetractPalletClose:
GVL_IO.LD_YPalletCloseExtend := FALSE;
GVL_IO.LD_YPalletCloseRetract := TRUE;
END_ACTION

METHOD PUBLIC AssignStationStatusForHMI : BOOL
VAR_INPUT
END_VAR
Status.StationsState[MM_CONST.LOAD_1_STA_HMI_STATE] := State;
IF (NOT LotsData.Lot.RejectUnloadEnabled) THEN
	Status.StationStauts[MM_CONST.LOAD_1_STA_HMI_STATE] := OverallStationStatus.eDisabled;
ELSE 
	CASE State OF 
	eLoadSta1State.eUnknown,eLoadSta1State.eError,eLoadSta1State.ePalletReleaseLowered:
		Status.StationStauts[MM_CONST.LOAD_1_STA_HMI_STATE] := OverallStationStatus.eError;
    eLoadSta1State.eInit,
	eLoadSta1State.eHoming:
	    Status.StationStauts[MM_CONST.LOAD_1_STA_HMI_STATE] := OverallStationStatus.eHoming;
		
	eLoadSta1State.eReady:
	     Status.StationStauts[MM_CONST.LOAD_1_STA_HMI_STATE] := OverallStationStatus.eWaitingForParts;
		 
	eLoadSta1State.eWaitForIBTrackClear:
	       Status.StationStauts[MM_CONST.LOAD_1_STA_HMI_STATE] := OverallStationStatus.eWarning;
		   
    
	eLoadSta1State.ePalletHoldDownEngage,
	eLoadSta1State.ePalletHoldDownEngaged,
	eLoadSta1State.ePalletReleaseRaise,
	eLoadSta1State.ePalletReleaseRaised,
	eLoadSta1State.eWaitForYushinPrepareLoad,
	eLoadSta1State.eWaitForYushinToolDown,	
	eLoadSta1State.ePalletReleaseLower,
	eLoadSta1State.eWaitForYushinToolUp,	
	eLoadSta1State.eProcessing:
	     Status.StationStauts[MM_CONST.LOAD_1_STA_HMI_STATE] := OverallStationStatus.eRunning;
		 
	eLoadSta1State.eStopActive:
	     Status.StationStauts[MM_CONST.LOAD_1_STA_HMI_STATE] := OverallStationStatus.eCycleStop;
    	
	ELSE;	
	END_CASE

END_IF

Status.StationStauts[MM_CONST.LOAD_2_STA_HMI_STATE] := Status.StationStauts[MM_CONST.LOAD_1_STA_HMI_STATE];
Status.StationStauts[MM_CONST.LOAD_3_STA_HMI_STATE] := Status.StationStauts[MM_CONST.LOAD_1_STA_HMI_STATE];
Status.StationStauts[MM_CONST.LOAD_4_STA_HMI_STATE] := Status.StationStauts[MM_CONST.LOAD_1_STA_HMI_STATE];
END_METHOD

METHOD PUBLIC ClearVehicleTrigger : BOOL
VAR_INPUT
END_VAR
xTrigger := FALSE;
CycleNumb :=0;
LoadingComplete:= FALSE;
HoldVehicleAtIBStop := FALSE;
END_METHOD

PROPERTY PUBLIC HoldVehicle_IBStop : BOOL
GET
HoldVehicle_IBStop := HoldVehicleAtIBStop;
END_GET
END_PROPERTY

METHOD PUBLIC IsFaulted : BOOL
VAR_INPUT
END_VAR
IsFaulted := (State = eLoadSta1State.eUnknown OR State = eLoadSta1State.eError);
END_METHOD

METHOD PUBLIC IsInboundTrackClear : BOOL
VAR_INPUT
END_VAR
VAR
	byCounter :BYTE;
	VehicleInRobotInboundPath: BOOL;
	KeepOffStartPOS: REAL;
	KeepOffStopPOS: REAL;
END_VAR
IsInboundTrackClear := TRUE;
KeepOffStartPos := MM_CONST.IB_STOP_ROBOT_CLEAR_POS+ (MM_CONST.Vehicle_Length)/1000;
KeepOffStopPos	:= MM_CONST.CAP_POS - (MM_CONST.Vehicle_Length*2/1000);
FOR byCounter := 1 TO MM_CONST.MAX_VEHICLES BY 1 DO  // if there is any vehicle in the Inbound track, do not load any parts
	IF ((STATUS.MMVehiclesStatus[byCounter].VehiclePos > KeepOffStartPos) AND (STATUS.MMVehiclesStatus[byCounter].VehiclePos < KeepOffStopPos)) THEN
		IsInboundTrackClear := FALSE;
	END_IF
END_FOR
END_METHOD

METHOD PUBLIC IsLoadWaitingForYushin : BOOL
VAR_INPUT
END_VAR
IsLoadWaitingForYushin := (State = eLoadSta1State.eWaitForYushinPrepareLoad);
END_METHOD

METHOD PUBLIC IsPalletCloseExtended : BOOL
VAR_INPUT
END_VAR
IsPalletCloseExtended := (GVL_IO.LD_XPalletCloseExtended_1_2 AND GVL_IO.LD_XPalletCloseExtended_3_4
                          AND NOT GVL_IO.LD_XPalletCloseRetracted_1_2 AND NOT  GVL_IO.LD_XPalletCloseRetracted_3_4);
IF(NOT IsPalletCloseExtended ) THEN
	Status.Load1StatusMsg:= 'Load: Check Pallet Close Sensors';
END_IF
END_METHOD

METHOD PUBLIC IsPalletCloseRetracted : BOOL
VAR_INPUT
END_VAR
IsPalletCloseRetracted := (NOT GVL_IO.LD_XPalletCloseExtended_1_2 AND GVL_IO.LD_XPalletCloseRetracted_1_2
                          AND NOT GVL_IO.LD_XPalletCloseExtended_3_4 AND GVL_IO.LD_XPalletCloseRetracted_3_4);
IF(NOT IsPalletCloseRetracted ) THEN
	Status.Load1StatusMsg:= 'Load: Check Pallet Close Sensors';
END_IF
END_METHOD

METHOD PUBLIC IsPalletHoldDownEngaged : BOOL
VAR_INPUT
END_VAR
IsPalletHoldDownEngaged := (GVL_IO.LD_XPalletHoldRetractEngage AND NOT GVL_IO.LD_XPalletHoldDownExtendHome);
IF(NOT IsPalletHoldDownEngaged) THEN
	Status.Load1StatusMsg:= 'Load: Check Pallet Hold Down';
END_IF
END_METHOD

METHOD PUBLIC IsPalletHoldDownFree : BOOL
VAR_INPUT
END_VAR
IsPalletHoldDownFree := (NOT GVL_IO.LD_XPalletHoldRetractEngage AND GVL_IO.LD_XPalletHoldDownExtendHome);
IF(NOT IsPalletHoldDownFree) THEN
	Status.Load1StatusMsg:= 'Load: Check Pallet Hold Down';
END_IF
END_METHOD

METHOD PUBLIC IsPalletReleaseEngaged : BOOL
VAR_INPUT
END_VAR
IsPalletReleaseEngaged := (NOT GVL_IO.LD_XPalletReleaseHome AND GVL_IO.LD_XPalletReleaseExtended); 
IF(NOT IsPalletReleaseEngaged) THEN
	Status.Load1StatusMsg:= 'Load: Check Pallet Release';
END_IF
END_METHOD

METHOD IsPalletReleaseFree : BOOL
VAR_INPUT
END_VAR
IsPalletReleaseFree := (GVL_IO.LD_XPalletReleaseHome AND NOT GVL_IO.LD_XPalletReleaseExtended); 
IF(NOT IsPalletReleaseFree) THEN
	Status.Load1StatusMsg:= 'Load: Check Pallet Release';
END_IF
END_METHOD

PROPERTY PUBLIC LoadComplete : BOOL
SET
LoadingComplete := LoadComplete;
END_SET
END_PROPERTY

PROPERTY PUBLIC Ready : BOOL
GET
Ready := (State = eLoadSta1State.eReady);
END_GET
END_PROPERTY

ACTION ResetDwellTimer:
DwellTimer(IN:= FALSE);
END_ACTION

METHOD PUBLIC ResetState : BOOL
VAR_INPUT
END_VAR
	State := eLoadSta1State.eUnknown;
	NextState := eLoadSta1State.eUnknown;
END_METHOD

ACTION ResetStateTimer:
StateTimer(IN:= FALSE);
END_ACTION

PROPERTY PUBLIC Trigger : BOOL
SET
xTrigger := Trigger;
END_SET
END_PROPERTY

METHOD PUBLIC UpdatePartData : BOOL
VAR_INPUT	
END_VAR
VAR
	
END_VAR
memset(ADR(PartsData.Status[VUT]),0,SIZEOF(PartDataType));
PartsData.Status[VUT].LoadTime := SYSTEMTIME_TO_STRING(Logging.fbCurrTime.systemTime);
PartsData.Status[VUT].CavityNumber := RowNumber + SeedNumber;
CycleNumb := CycleNumb+1; // Use this till Yushin Robot sends out this information with Bit Location ID
PartsData.Status[VUT].OverallStatus := ePartStatus.eLoaded; // At least that is the assumption. We may want to check on how to turn off cavities later, but this will be caught by vision.
PartsData.Status[VUT].BarrelSize := LotsData.Lot.BarrelSize; // we are copying this data in case we might in future want to have more than one lots running at the same time on the machine
PartsData.Status[VUT].PartNumber := LotsData.Lot.PartNumber; // we are copying this data in case we might in future want to have more than one lots running at the same time on the machine
PartsData.Status[VUT].LotNumber := LotsData.Lot.LotNumber; // we are copying this data in case we might in future want to have more than one lots running at the same time on the machine
END_METHOD

PROPERTY PUBLIC VehicleUnderTest : BYTE
GET
VehicleUnderTest := VUT;
END_GET
SET
VUT := VehicleUnderTest;
END_SET
END_PROPERTY

END_FUNCTION_BLOCK

// ---- POUs/Load2Station.TcPOU
FUNCTION_BLOCK PUBLIC Load2Station
VAR_INPUT
END_VAR
VAR_OUTPUT
END_VAR
VAR
	xTrigger :BOOL := FALSE; // triggers processing
	State : eLoadSta2State := eLoadSta2State.eUnknown;
	NextState : eLoadSta2State := eLoadSta2State.eUnknown;
	bFirst : BOOL := TRUE;
	VUT : BYTE; //VehicleID Under Station
	DwellTimer : TON;
	LoadingComplete : BOOL := FALSE;
	CycleNumb: INT :=0;
	RowNumber :INT:=0;
	SeedNumber : INT:=9;
END_VAR

IF (GVL_IO.MachineEStopped) THEN 
	State := eLoadSta2State.eUnknown;
	NextState := eLoadSta2State.eUnknown;
END_IF

CASE State OF
eLoadSta2State.eUnknown:
	NextState := eLoadSta2State.eReady;

eLoadSta2State.eInit:

eLoadSta2State.eHoming:

eLoadSta2State.eReady:

   IF (xTrigger) THEN
		NextState := eLoadSta2State.eWaitForLoadComplete;
		
		DwellTimer(IN:=FALSE);		
	END_IF

eLoadSta2State.eDwell:

eLoadSta2State.eWaitForLoadComplete:
	 IF (LoadingComplete) THEN
		NextState := eLoadSta2State.eDepart;
        UpdatePartData();		
		LoadingComplete := FALSE;
		DwellTimer(IN:=FALSE);
	END_IF


eLoadSta2State.eProcessing:

eLoadSta2State.eDepart:
  	Stations.fbRoutePlanner.M_NotifyVehStaCmpl(StationIndex:= MM_CONST.LOAD_2_STA, VehicleID := VUT);
	xTrigger := FALSE;
	IF (Stations.fbCycleControl.StopRequested) THEN
		NextState := eLoadSta2State.eStopActive;
	ELSE	
		NextState := eLoadSta2State.eReady;	
	END_IF
	
eLoadSta2State.eStopActive:
	IF (NOT Stations.fbCycleControl.StopRequested) THEN
		NextState := eLoadSta2State.eReady;
	END_IF;
	
eLoadSta2State.eError:

END_CASE

IF (State <> NextState) THEN
	bFirst := TRUE;
ELSE
	bFirst := FALSE;
END_IF

State := NextState;
Status.StationsState[MM_CONST.LOAD_2_STA_HMI_STATE] := State;

METHOD PUBLIC ClearVehicleTrigger : BOOL
VAR_INPUT
END_VAR
xTrigger := FALSE;
END_METHOD

PROPERTY PUBLIC LoadComplete : BOOL
SET
LoadingComplete := LoadComplete;
END_SET
END_PROPERTY

METHOD PUBLIC ResetState : BOOL
VAR_INPUT
END_VAR
State := eLoadSta2State.eUnknown;
NextState := eLoadSta2State.eUnknown;
END_METHOD

METHOD PUBLIC SetRowNumber : BOOL
VAR_INPUT
	RowLocationNumber : INT;
END_VAR
RowNumber := RowLocationNumber;
END_METHOD

PROPERTY PUBLIC Trigger : BOOL
SET
xTrigger := Trigger;
END_SET
END_PROPERTY

METHOD PUBLIC UpdatePartData : BOOL
VAR_INPUT
END_VAR
memset(ADR(PartsData.Status[VUT]),0,SIZEOF(PartDataType));
PartsData.Status[VUT].LoadTime := SYSTEMTIME_TO_STRING(Logging.fbCurrTime.systemTime);
//PartsData.Status[VUT].CavityNumber := 5 + (CycleNumb MOD 4);
PartsData.Status[VUT].CavityNumber := RowNumber + SeedNumber;
CycleNumb := CycleNumb+1; // Use this till Yushin Robot sends out this information with Bit Location ID
PartsData.Status[VUT].OverallStatus := ePartStatus.eLoaded; // At least that is the assumption. We may want to check on how to turn off cavities later, but this will be caught by vision.
PartsData.Status[VUT].BarrelSize := LotsData.Lot.BarrelSize; // we are copying this data in case we might in future want to have more than one lots running at the same time on the machine
PartsData.Status[VUT].PartNumber := LotsData.Lot.PartNumber; // we are copying this data in case we might in future want to have more than one lots running at the same time on the machine
PartsData.Status[VUT].LotNumber := LotsData.Lot.LotNumber; // we are copying this data in case we might in future want to have more than one lots running at the same time on the machine
END_METHOD

PROPERTY PUBLIC VehicleUnderTest : BYTE
GET
VehicleUnderTest := VUT;
END_GET
SET
VUT := VehicleUnderTest;
END_SET
END_PROPERTY

END_FUNCTION_BLOCK

// ---- POUs/Load3Station.TcPOU
FUNCTION_BLOCK PUBLIC Load3Station
VAR_INPUT
END_VAR
VAR_OUTPUT
END_VAR
VAR
	xTrigger :BOOL := FALSE; // triggers processing
	State : eLoadSta3State := eLoadSta3State.eUnknown;
	NextState : eLoadSta3State := eLoadSta3State.eUnknown;
	bFirst : BOOL := TRUE;
	VUT : BYTE; //VehicleID Under Station
	DwellTimer : TON;
	LoadingComplete : BOOL := FALSE;
	CycleNumb: INT := 0;
	RowNumber :INT:=0;
	SeedNumber : INT:=5;
END_VAR

IF (GVL_IO.MachineEStopped) THEN 
	State := eLoadSta3State.eUnknown;
	NextState := eLoadSta3State.eUnknown;
END_IF

CASE State OF
eLoadSta3State.eUnknown:
	NextState := eLoadSta3State.eReady;

eLoadSta3State.eInit:

eLoadSta3State.eHoming:

eLoadSta3State.eReady:

IF (xTrigger) THEN
		NextState := eLoadSta3State.eWaitForLoadComplete;
		
		DwellTimer(IN:=FALSE);	
	END_IF

eLoadSta3State.eDwell:

eLoadSta3State.eWaitForLoadComplete:
	 IF (LoadingComplete) THEN
		NextState := eLoadSta3State.eDepart;
		UpdatePartData();
		LoadingComplete := FALSE;
		DwellTimer(IN:=FALSE);
	END_IF


eLoadSta3State.eProcessing:

eLoadSta3State.eDepart:
	Stations.fbRoutePlanner.M_NotifyVehStaCmpl(StationIndex:= MM_CONST.LOAD_3_STA, VehicleID := VUT);
	xTrigger := FALSE;
    IF (Stations.fbCycleControl.StopRequested) THEN
		NextState := eLoadSta3State.eStopActive;
	ELSE	
		NextState := eLoadSta3State.eReady;	
	END_IF

eLoadSta3State.eStopActive:
	IF (NOT Stations.fbCycleControl.StopRequested) THEN
		NextState := eLoadSta3State.eReady;
	END_IF
	
eLoadSta3State.eError:

END_CASE

IF (State <> NextState) THEN
	bFirst := TRUE;
ELSE
	bFirst := FALSE;
END_IF

State := NextState;
Status.StationsState[MM_CONST.LOAD_3_STA_HMI_STATE] := State;

METHOD PUBLIC ClearVehicleTrigger : BOOL
VAR_INPUT
END_VAR
xTrigger := FALSE;
END_METHOD

PROPERTY PUBLIC LoadComplete : BOOL
SET
LoadingComplete := LoadComplete;
END_SET
END_PROPERTY

METHOD PUBLIC ResetState : BOOL
VAR_INPUT
END_VAR
	State := eLoadSta3State.eUnknown;
	NextState := eLoadSta3State.eUnknown;
END_METHOD

METHOD PUBLIC SetRowNumber : BOOL
VAR_INPUT
	RowLocationNumber : INT;
END_VAR
RowNumber := RowLocationNumber;
END_METHOD

PROPERTY PUBLIC Trigger : BOOL
SET
xTrigger := Trigger;
END_SET
END_PROPERTY

METHOD PUBLIC UpdatePartData : BOOL
VAR_INPUT
END_VAR
memset(ADR(PartsData.Status[VUT]),0,SIZEOF(PartDataType));
PartsData.Status[VUT].LoadTime := SYSTEMTIME_TO_STRING(Logging.fbCurrTime.systemTime);
//PartsData.Status[VUT].CavityNumber := 9 + (CycleNumb MOD 4);
PartsData.Status[VUT].CavityNumber := RowNumber + SeedNumber;
CycleNumb := CycleNumb+1; // Use this till Yushin Robot sends out this information with Bit Location ID
PartsData.Status[VUT].OverallStatus := ePartStatus.eLoaded; // At least that is the assumption. We may want to check on how to turn off cavities later, but this will be caught by vision.
PartsData.Status[VUT].BarrelSize := LotsData.Lot.BarrelSize; // we are copying this data in case we might in future want to have more than one lots running at the same time on the machine
PartsData.Status[VUT].PartNumber := LotsData.Lot.PartNumber; // we are copying this data in case we might in future want to have more than one lots running at the same time on the machine
PartsData.Status[VUT].LotNumber := LotsData.Lot.LotNumber; // we are copying this data in case we might in future want to have more than one lots running at the same time on the machine
END_METHOD

PROPERTY PUBLIC VehicleUnderTest : BYTE
GET
VehicleUnderTest := VUT;
END_GET
SET
VUT := VehicleUnderTest;
END_SET
END_PROPERTY

END_FUNCTION_BLOCK

// ---- POUs/Load4Station.TcPOU
FUNCTION_BLOCK Load4Station
VAR_INPUT
END_VAR
VAR_OUTPUT
END_VAR
VAR
	xTrigger :BOOL := FALSE; // triggers processing
	State : eLoadSta4State := eLoadSta4State.eUnknown;
	NextState : eLoadSta4State := eLoadSta4State.eUnknown;
	bFirst : BOOL := TRUE;
	VUT : BYTE; //VehicleID Under Station
	DwellTimer : TON;
	LoadingComplete : BOOL := FALSE;
	CycleNumb: INT := 0;
	RowNumber :INT:=0;
	SeedNumber : INT:=1;
END_VAR

IF (GVL_IO.MachineEStopped) THEN 
	State := eLoadSta4State.eUnknown;
	NextState := eLoadSta4State.eUnknown;
END_IF

CASE State OF

eLoadSta4State.eUnknown:
	NextState := eLoadSta4State.eReady;

eLoadSta4State.eInit:

eLoadSta4State.eHoming:

eLoadSta4State.eReady:

	IF (xTrigger) THEN
		NextState := eLoadSta4State.eWaitForLoadComplete;
		
		DwellTimer(IN:=FALSE);		
	END_IF

eLoadSta4State.eDwell:


eLoadSta4State.eWaitForLoadComplete:
	 IF (LoadingComplete) THEN
		NextState := eLoadSta4State.eDepart;
		UpdatePartData();
		LoadingComplete := FALSE;
		DwellTimer(IN:=FALSE);
	END_IF
	
eLoadSta4State.eProcessing:


eLoadSta4State.eDepart:
	Stations.fbRoutePlanner.M_NotifyVehStaCmpl(StationIndex:= MM_CONST.LOAD_4_STA, VehicleID := VUT);
	xTrigger := FALSE;
    IF (Stations.fbCycleControl.StopRequested) THEN
		NextState := eLoadSta4State.eStopActive;
	ELSE	
		NextState := eLoadSta4State.eReady;	
	END_IF

eLoadSta4State.eStopActive:
	IF (NOT Stations.fbCycleControl.StopRequested) THEN
		NextState := eLoadSta4State.eReady;
	END_IF

eLoadSta4State.eError:

END_CASE

IF (State <> NextState) THEN
	bFirst := TRUE;
ELSE
	bFirst := FALSE;
END_IF

State := NextState;
Status.StationsState[MM_CONST.LOAD_4_STA_HMI_STATE] := State;

METHOD PUBLIC ClearVehicleTrigger : BOOL
VAR_INPUT
END_VAR
xTrigger := FALSE;
END_METHOD

PROPERTY PUBLIC LoadComplete : BOOL
SET
LoadingComplete := LoadComplete;
END_SET
END_PROPERTY

METHOD PUBLIC ResetState : BOOL
VAR_INPUT
END_VAR
	State := eLoadSta4State.eUnknown;
	NextState := eLoadSta4State.eUnknown;
END_METHOD

METHOD PUBLIC SetRowNumber : BOOL
VAR_INPUT
	RowLocationNumber : INT;
END_VAR
RowNumber := RowLocationNumber;
END_METHOD

PROPERTY PUBLIC Trigger : BOOL
SET
xTrigger := Trigger;
END_SET
END_PROPERTY

METHOD PUBLIC UpdatePartData : BOOL
VAR_INPUT
END_VAR
memset(ADR(PartsData.Status[VUT]),0,SIZEOF(PartDataType));
PartsData.Status[VUT].LoadTime := SYSTEMTIME_TO_STRING(Logging.fbCurrTime.systemTime);
//PartsData.Status[VUT].CavityNumber := 13 + (CycleNumb MOD 4);
PartsData.Status[VUT].CavityNumber := RowNumber + SeedNumber;
CycleNumb := CycleNumb+1; // Use this till Yushin Robot sends out this information with Bit Location ID
PartsData.Status[VUT].OverallStatus := ePartStatus.eLoaded; // At least that is the assumption. We may want to check on how to turn off cavities later, but this will be caught by vision.
PartsData.Status[VUT].BarrelSize := LotsData.Lot.BarrelSize; // we are copying this data in case we might in future want to have more than one lots running at the same time on the machine
PartsData.Status[VUT].PartNumber := LotsData.Lot.PartNumber; // we are copying this data in case we might in future want to have more than one lots running at the same time on the machine
PartsData.Status[VUT].LotNumber := LotsData.Lot.LotNumber; // we are copying this data in case we might in future want to have more than one lots running at the same time on the machine
END_METHOD

PROPERTY PUBLIC VehicleUnderTest : BYTE
GET
VehicleUnderTest := VUT;
END_GET
SET
VUT := VehicleUnderTest;
END_SET
END_PROPERTY

END_FUNCTION_BLOCK

// ---- POUs/OB_StopRobotClearStation.TcPOU
FUNCTION_BLOCK PUBLIC OB_StopRobotClearStation
VAR_INPUT
END_VAR
VAR_OUTPUT
END_VAR
VAR
	xTrigger :BOOL := FALSE; // triggers processing
	State : eOB_StopRobotClearStaState := eOB_StopRobotClearStaState.eUnknown;
	NextState : eOB_StopRobotClearStaState := eOB_StopRobotClearStaState.eUnknown;
	bFirst : BOOL := TRUE;
	VUT : BYTE; //VehicleID Under Station
	DwellTimer : TON;
	MoveVehicleToLoad: BOOL := TRUE; //We have to send the Vehicle to Load Position # 4 at startup
END_VAR

CASE State OF

eOB_StopRobotClearStaState.eUnknown:
	NextState := eOB_StopRobotClearStaState.eReady;

eOB_StopRobotClearStaState.eInit:

eOB_StopRobotClearStaState.eHoming:

eOB_StopRobotClearStaState.eReady:
IF (xTrigger) THEN
		NextState := eOB_StopRobotClearStaState.eProcessing;
		
		DwellTimer(IN:=FALSE);
	END_IF

eOB_StopRobotClearStaState.eDwell:

eOB_StopRobotClearStaState.eProcessing:
  IF (MoveVehicleToLoad) THEN
	  NextState := eOB_StopRobotClearStaState.eDepart;
  END_IF

eOB_StopRobotClearStaState.eDepart:
	
    Stations.fbRoutePlanner.M_NotifyVehStaCmpl(StationIndex:= MM_CONST.OB_STOP_ROBOT_CLEAR_STA, VehicleID := VUT);
	xTrigger := FALSE;
	MoveVehicleToLoad := FALSE;	
	NextState := eOB_StopRobotClearStaState.eReady;

eOB_StopRobotClearStaState.eError:

ELSE;

END_CASE

IF (State <> NextState) THEN
	bFirst := TRUE;
ELSE
	bFirst := FALSE;
END_IF

State := NextState;

Status.StationsState[MM_CONST.OB_STOP_ROBOT_CLEAR_STA_HMI_STATE] := State;

METHOD PUBLIC ClearVehicleTrigger : BOOL
VAR_INPUT
END_VAR
xTrigger := FALSE;
State := eOB_StopRobotClearStaState.eUnknown;
NextState:= eOB_StopRobotClearStaState.eUnknown;
bFirst  := TRUE;
MoveVehicleToLoad := TRUE; //We have to send the Vehicle to Load Position # 4 at startup
END_METHOD

PROPERTY PUBLIC MoveToLoading : BOOL
SET
MoveVehicleToLoad := MoveToLoading;
END_SET
END_PROPERTY

PROPERTY PUBLIC Trigger : BOOL
SET
xTrigger := Trigger;
END_SET
END_PROPERTY

PROPERTY PUBLIC VehicleUnderTest : BYTE
GET
VehicleUnderTest := VUT;
END_GET
SET
VUT := VehicleUnderTest;
END_SET
END_PROPERTY

END_FUNCTION_BLOCK

// ---- POUs/OB_StopBeforeVisionStation.TcPOU
FUNCTION_BLOCK PUBLIC OB_StopBeforeVisionStation
VAR_INPUT
END_VAR
VAR_OUTPUT
END_VAR
VAR
	xTrigger :BOOL := FALSE; // triggers processing
	State : eOB_StopBeforeVisionState := eOB_StopBeforeVisionState.eUnknown;
	NextState : eOB_StopBeforeVisionState := eOB_StopBeforeVisionState.eUnknown;
	bFirst : BOOL := TRUE;
	VUT : BYTE; //VehicleID Under Station
	DwellTimer : TON;
END_VAR

CASE State OF

eOB_StopBeforeVisionState.eUnknown:
	NextState := eOB_StopBeforeVisionState.eReady;

eOB_StopBeforeVisionState.eInit:

eOB_StopBeforeVisionState.eHoming:

eOB_StopBeforeVisionState.eReady:
	IF (xTrigger) THEN
		NextState := eOB_StopBeforeVisionState.eDwell;		
		DwellTimer(IN:=FALSE);
	END_IF

eOB_StopBeforeVisionState.eDwell:
	DwellTimer(IN:=TRUE, PT := T#600MS);
	IF (GVL_IO.VS_XPartPresentBeforeVision) THEN 
		PartsData.Status[VUT].OverallStatus := ePartStatus.eLoaded;
        NextState := eOB_StopBeforeVisionState.eProcessing;		
		DwellTimer(IN:=FALSE);
	END_IF
	IF (DwellTimer.Q) THEN // just call it loaded, no sensor is present 
		NextState := eOB_StopBeforeVisionState.eProcessing;		
		PartsData.Status[VUT].OverallStatus := ePartStatus.eLoaded;
		DwellTimer(IN:=FALSE);
	END_IF

eOB_StopBeforeVisionState.eProcessing:
	IF (NOT Stations.fbVisionSta.InspectionOnGoing) THEN
		NextState := eOB_StopBeforeVisionState.eDepart;
	END_IF

eOB_StopBeforeVisionState.eDepart:
	    UpdatePartData();
		Stations.fbRoutePlanner.M_NotifyVehStaCmpl(StationIndex:= MM_CONST.STOP_BEFORE_VISION_STA, VehicleID := VUT);
		xTrigger := FALSE;
		NextState := eOB_StopBeforeVisionState.eReady;

eOB_StopBeforeVisionState.eError:
END_CASE

IF (State <> NextState) THEN
	bFirst := TRUE;
ELSE
	bFirst := FALSE;
END_IF

State := NextState;

METHOD PUBLIC ClearVehicleTrigger : BOOL
VAR_INPUT
END_VAR
xTrigger := FALSE;
END_METHOD

PROPERTY PUBLIC Trigger : BOOL
SET
xTrigger := Trigger;
END_SET
END_PROPERTY

METHOD PUBLIC UpdatePartData : BOOL
VAR_INPUT
END_VAR
PartsData.Status[VUT].BurnOffTemp := GVL_IO.BU_Temperature/10;
END_METHOD

PROPERTY PUBLIC VehicleUnderTest : BYTE
GET
VehicleUnderTest := VUT;
END_GET
SET
VUT := VehicleUnderTest;
END_SET
END_PROPERTY

END_FUNCTION_BLOCK

// ---- POUs/VisionStation.TcPOU
FUNCTION_BLOCK PUBLIC VisionStation
VAR_INPUT
END_VAR
VAR_OUTPUT
END_VAR
VAR
	xTrigger :BOOL := FALSE; // triggers processing
	State : eVisionStaState := eVisionStaState.eUnknown;
	NextState : eVisionStaState := eVisionStaState.eUnknown;
	ErrorReturnState : eVisionStaState := eVisionStaState.eUnknown;
	bFirst : BOOL := TRUE;
	VUT : BYTE; //VehicleID Under Station
	DwellTimer : TON;
	StateTimer : TON;
	VehicleStopTime : TIME := T#150MS; //was 75ms, believed to cause duplicate bad info 3-20-19 CMS
	SDNumber : BYTE;
	ProgramNumber : BYTE;
END_VAR

// Sequence of events:
// Check if Cmd is Ready to Process else, give message to operator
// Check if Correct Program in loaded, else change to correct program for Barrel Type
// Check if in Run Mode, else put in Run Mode
// Check if all Cameras are ready to accept triggers, else reset Triggers
// Go to Wait for Vehicle Trigger
// Complete Inspection
// Depart vehicle and go to state where we check if all cameras are ready to accept triggers


IF (GVL_IO.MachineEStopped) THEN 
	State := eVisionStaState.eUnknown;
	NextState := eVisionStaState.eUnknown;
	ErrorReturnState := eVisionStaState.eUnknown;
	Status.VisionStatusMsg:= 'Vision  Unknown, Check AIR, E-STOP and Hit Start';
END_IF

CASE State OF
	
eVisionStaState.eUnknown:
	GVL_IO.VS_YBarrelLED := FALSE; 
	GVL_IO.VS_YTrigger1  := FALSE;
	GVL_IO.VS_YTrigger2  := FALSE;
	GVL_IO.VS_YTrigger3  := FALSE;
	GVL_IO.VS_YTrigger4  := FALSE;
	GVL_IO.VS_YCmdRequest := FALSE;
	GVL_IO.VS_YResultAck := TRUE;
	GVL_IO.VS_YErrorReset := FALSE;
	
	IF (GVL_IO.MC_XStartPB AND GVL_IO.MC_NotEStopped) THEN //Vision Sta doesn't need Air Pressure for debug, so removed Air Pressure Check
		NextState := eVisionStaState.eInit; //eVisionStaState.eCheckToolPosition; // ;	
	END_IF	


eVisionStaState.eCheckToolPosition:	
	IF (LotsData.Lot.BarrelSize = eBarrelType.Size55cc) THEN
		IF (GVL_IO.VS_XToolingLocationUpper AND GVL_IO.VS_XToolingLocationLower) THEN
			 NextState := eVisionStaState.eInit;
		ELSE
			ErrorReturnState := eVisionStaState.eCheckToolPosition;
            NextState := eVisionStaState.eError;
        	Status.VisionStatusMsg:= 'Vision: Incorrect 55cc ToolID,Fix and Hit Start';
		END_IF
	ELSIF (LotsData.Lot.BarrelSize = eBarrelType.Size30cc) THEN
		IF (NOT GVL_IO.VS_XToolingLocationUpper AND GVL_IO.VS_XToolingLocationLower) THEN
			 NextState := eVisionStaState.eInit;
		ELSE
			ErrorReturnState := eVisionStaState.eCheckToolPosition;
            NextState := eVisionStaState.eError;
        	Status.VisionStatusMsg:= 'Vision: Incorrect 30cc ToolID,Fix and Hit Start';
		END_IF
	ELSE
	     ErrorReturnState := eVisionStaState.eUnknown;
         NextState := eVisionStaState.eError;
         Status.VisionStatusMsg:= 'Vision: Incorrect Part Selection, Start New Lot';
	END_IF
	
eVisionStaState.eInit:
     GVL_IO.VS_YBarrelLED := FALSE;
	 GVL_IO.VS_YTrigger1  := FALSE;
	 GVL_IO.VS_YTrigger2  := FALSE;
	 GVL_IO.VS_YTrigger3  := FALSE;
	 GVL_IO.VS_YTrigger4  := FALSE;
	 GVL_IO.VS_YCmdRequest := FALSE;
	 GVL_IO.VS_YResultAck  := TRUE;
	 GVL_IO.VS_YErrorReset := FALSE;
	IF (GVL_IO.VS_XError) THEN
		GVL_IO.VS_YErrorReset := TRUE;		
    END_IF 
	DwellTimer(IN:=TRUE, PT:= T#2S);
	IF (DwellTimer.Q) THEN
		DwellTimer(IN:=FALSE);
		GVL_IO.VS_YResultAck  := FALSE;
		GVL_IO.VS_YErrorReset := FALSE;		
		IF(GVL_IO.VS_XCmdReady AND NOT GVL_IO.VS_XBusy AND NOT GVL_IO.VS_XError) THEN
			NextState := eVisionStaState.eHoming;				
		ELSE 
			NextState := eVisionStaState.eCmdTriggerReset;
		END_IF
	END_IF
	
eVisionStaState.eCmdTriggerReset:
	GVL_IO.VS_YCmdNumber := 15;
	IF (GVL_IO.VS_XCmdReady) THEN
		DwellTimer(IN:=TRUE, PT:=T#50MS);
		IF (DwellTimer.Q) THEN
			DwellTimer(IN:=FALSE);
			GVL_IO.VS_YCmdRequest := TRUE;
			NextState := eVisionStaState.eCheckTriggerResetCmpl;
			StateTimer(IN:=FALSE);
		END_IF	
	ELSE
		NextState := eVisionStaState.eError;
		ErrorReturnState := eVisionStaState.eUnknown;
        Status.VisionStatusMsg:= 'Vision: Keyence Not Ready, fix in Keyence HMI, then Press Start';
	END_IF

eVisionStaState.eCheckTriggerResetCmpl:
	IF (GVL_IO.VS_XCmdCmpl) THEN
		GVL_IO.VS_YCmdRequest := FALSE;
		NextState := eVisionStaState.eError;
		ErrorReturnState := eVisionStaState.eInit;
		Status.VisionStatusMsg:= 'Vision System remotely reset by PLC, Press Start to continue';
	END_IF

	
eVisionStaState.eHoming: // get program that is correct loaded 
    IF (GVL_IO.VS_XReady1 AND GVL_IO.VS_XReady2 AND GVL_IO.VS_XReady3 AND GVL_IO.VS_XReady4) THEN
		NextState := eVisionStaState.eConfirmRunState;
	ELSE
		NextState := eVisionStaState.eUnknown;
		Status.VisionStatusMsg:= 'Vision not Ready, check if Keyence Controller is ready/run mode';
		DwellTimer(IN:=FALSE);
	END_IF


	
eVisionStaState.eConfirmRunState:
     IF (GVL_IO.VS_XRun) THEN 
		 NextState := eVisionStaState.eGetProgramNumber;
		 DwellTimer(IN:=FALSE);
	 END_IF
	 Status.VisionStatusMsg:= 'Put Vision Station in Run Mode';
 /// Here we need to put the controller in the Run State either programatically and tell the operator to put in  RUN state... execute the control parameter write 
 
eVisionStaState.eGetProgramNumber:
//Check if cmd ready
//Send read command
	IF(GVL_IO.VS_XCmdReady) THEN
		GVL_IO.VS_YCmdNumber := VIS_CONST.Cmd_ReadProgram; //write command number
		GVL_IO.VS_YCmdParam1 := 0;    //write parameters
		GVL_IO.VS_YCmdParam2 := 0;
		GVL_IO.VS_YCmdRequest := TRUE;         //turn on command request flag

//check if command complete	
//read value
//cmd request flag off

	ELSIF (GVL_IO.VS_XCmdCmpl) THEN
		GVL_IO.VS_YCmdRequest := FALSE; 
		NextState := eVisionStaState.eCheckProgramNumber;
	END_IF

	
eVisionStaState.eCheckProgramNumber:
//compare to correct value
//if correct, next state
	SDNumber := GVL_IO.VS_XCmdData1;
	ProgramNumber := GVL_IO.VS_XCmdData2;
	
	IF((ProgramNumber = LotsData.Lot.VisionProgramNumber) AND (SDNumber = 1)) THEN
		NextState := eVisionStaState.eReady;
	ELSIF (LotsData.Lot.VisionStationRunSelect = eVisionEnableState.Disabled) THEN
		NextState := eVisionStaState.eReady;
ELSE	
		NextState := eVisionStaState.eChangeProgramNumber;
	END_IF

eVisionStaState.eChangeProgramNumber:
//check if cmd ready
//send change program cmd
	IF(GVL_IO.VS_XCmdReady) THEN
		GVL_IO.VS_YCmdNumber := VIS_CONST.Cmd_ChangeProgram; //write command number
		GVL_IO.VS_YCmdParam1 := 1;    //write parameters
		GVL_IO.VS_YCmdParam2 := DINT_TO_BYTE(LotsData.Lot.VisionProgramNumber);
		GVL_IO.VS_YCmdRequest := TRUE;         //turn on command request flag

//check if command complete	
//read value
//if 0 next state
//else Status.VisionStatusMsg 'Please select correct vision program manually'
	ELSIF (GVL_IO.VS_XCmdCmpl) THEN
		GVL_IO.VS_YCmdRequest := FALSE; 
		NextState := eVisionStaState.eGetProgramNumber;
		Status.VisionStatusMsg:= 'Please select correct vision program manually'; 	
	END_IF

	
eVisionStaState.eReady:
     GVL_IO.VS_YBarrelLED := TRUE;
	IF (xTrigger) THEN
		DwellTimer(IN:=TRUE, PT:= VehicleStopTime);
		IF (DwellTimer.Q) THEN			
			NextState := eVisionStaState.eBarellInspectTrigger;
			PartsData.Status[VUT].OverallStatus := ePartStatus.eReject; //define as reject upfront, later update status
			PartsData.Status[VUT].VisionInspectTime := SYSTEMTIME_TO_STRING(Logging.fbCurrTime.systemTime); // we are getting some empty time stamp
			DwellTimer(IN:=FALSE);
		END_IF
	END_IF
	GVL_IO.VS_YResultAck := FALSE;
	Status.VisionStatusMsg:= 'Waiting For Vehicle Trigger';

eVisionStaState.eWaitingForVehicleTrigger:

eVisionStaState.eBarellInspectTrigger:
    GVL_IO.VS_YTrigger2 := TRUE;
	GVL_IO.VS_YTrigger3 := TRUE;
	GVL_IO.VS_YTrigger4 := TRUE;
	//DwellTimer(IN:=TRUE, PT:= T#250MS);
	DwellTimer(IN:=TRUE, PT:= T#175MS);
	IF (DwellTimer.Q) THEN
		DwellTimer(IN:=FALSE);
		GVL_IO.VS_YTrigger1:=  FALSE;
		GVL_IO.VS_YTrigger2 := FALSE;
		GVL_IO.VS_YTrigger3 := FALSE;
		GVL_IO.VS_YTrigger4 := FALSE;
		GVL_IO.VS_YBarrelLED:= FALSE;
		NextState := eVisionStaState.eShortShotTrigger; //eVisionStaState.eWaitBarellInspectDone;
	END_IF

eVisionStaState.eShortShotTrigger:
     GVL_IO.VS_YTrigger1 := TRUE;
	 //DwellTimer(IN:=TRUE, PT:= T#250MS);
	 DwellTimer(IN:=TRUE, PT:= T#125MS);
	 IF (DwellTimer.Q) THEN
		 GVL_IO.VS_YTrigger1 := FALSE;
		 DwellTimer(IN:=FALSE);
		 NextState := eVisionStaState.eWaitShortShotDone;		 
	 END_IF

eVisionStaState.eWaitShortShotDone: 
// check the ACK bit here 
    GVL_IO.VS_YBarrelLED:= TRUE;
	DwellTimer(IN:=TRUE, PT:= T#10MS);
	IF (DwellTimer.Q) THEN
		NextState := eVisionStaState.eWaitBarellInspectDone;
		DwellTimer(IN:=FALSE);
	END_IF	

eVisionStaState.eWaitBarellInspectDone:
	DwellTimer(IN:=TRUE,PT:=T#10MS);
	IF (DwellTimer.Q) THEN
		IF (GVL_IO.VS_XReady1 AND GVL_IO.VS_XReady2 AND GVL_IO.VS_XReady3 AND GVL_IO.VS_XReady4) THEN
			NextState := eVisionStaState.eProcessVisionData;
			GVL_IO.VS_YTrigger1:=  FALSE;
			GVL_IO.VS_YTrigger2 := FALSE;
			GVL_IO.VS_YTrigger3 := FALSE;
			GVL_IO.VS_YTrigger4 := FALSE;
			//GVL_IO.VS_YBarrelLED:= FALSE;
			DwellTimer(IN:=FALSE);
        END_IF		
	END_IF

eVisionStaState.eProcessVisionData:
	DwellTimer(IN:=TRUE, PT:= T#200MS); //was 20ms, believed to cause duplicate bad info 3-20-19 CMS
	IF (DwellTimer.Q) THEN 
		DwellTimer(IN:=FALSE);	
		//PartsData.Status[VUT].OverallStatus := ePartStatus.eLoaded; // we know its not empty from initial check
		//PartsData.Status[VUT].OverallStatus := ePartStatus.eGoodPremium; // we need to remove this later 101717
	    UpdatePartData();
		GVL_IO.VS_YResultAck := TRUE;
  		NextState := eVisionStaState.eDepart;
	END_IF
   	 
	
eVisionStaState.eDepart:
	Stations.fbRoutePlanner.M_NotifyVehStaCmpl(StationIndex:= MM_CONST.VISION_STA, VehicleID := VUT);
	xTrigger := FALSE;
    IF (Stations.fbCycleControl.StopRequested) THEN
        NextState := eVisionStaState.eStopActive; 
    ELSE
		NextState := eVisionStaState.eConfirmRunState;
	END_IF
	
	

eVisionStaState.eStopActive:
 	IF (NOT Stations.fbCycleControl.StopRequested) THEN
		NextState := eVisionStaState.eConfirmRunState;
	END_IF
	Status.VisionStatusMsg:= 'Vision Cycle Stopped, hit START Button';
	GVL_IO.VS_YBarrelLED:= FALSE;
		
eVisionStaState.eError:
	IF (GVL_IO.MC_XStartPB) THEN
		NextState := ErrorReturnState;
		ErrorReturnState := eVisionStaState.eUnknown;
	END_IF


END_CASE

IF (State <> NextState) THEN
	bFirst := TRUE;
	StateTimer(IN:=FALSE);
ELSE
	bFirst := FALSE;
END_IF

State := NextState;

AssignStationStatusForHMI();

METHOD PUBLIC AssignStationStatusForHMI  : BOOL
VAR_INPUT
END_VAR
Status.StationsState[MM_CONST.VISION_STA_HMI_STATE] := State;
IF (LotsData.Lot.VisionStationRunSelect = eVisionEnableState.Disabled ) THEN
	Status.StationStauts[MM_CONST.VISION_STA_HMI_STATE] := OverallStationStatus.eDisabled;	
ELSE 
	CASE State OF 
	eVisionStaState.eUnknown, eVisionStaState.eError:
		Status.StationStauts[MM_CONST.VISION_STA_HMI_STATE] := OverallStationStatus.eError; 
    
    eVisionStaState.eInit, eVisionStaState.eHoming:
		Status.StationStauts[MM_CONST.VISION_STA_HMI_STATE] := OverallStationStatus.eHoming;
		
	eVisionStaState.eConfirmRunState,eVisionStaState.eGetProgramNumber,eVisionStaState.eCheckProgramNumber,eVisionStaState.eChangeProgramNumber:
	    Status.StationStauts[MM_CONST.VISION_STA_HMI_STATE] := OverallStationStatus.eWarning;
		
	eVisionStaState.eReady, eVisionStaState.eWaitingForVehicleTrigger:
	    Status.StationStauts[MM_CONST.VISION_STA_HMI_STATE] := OverallStationStatus.eWaitingForParts;
	
    eVisionStaState.eShortShotTrigger, eVisionStaState.eWaitShortShotDone,eVisionStaState.eBarellInspectTrigger,
	eVisionStaState.eWaitBarellInspectDone,eVisionStaState.eProcessVisionData:
	    Status.StationStauts[MM_CONST.VISION_STA_HMI_STATE] := OverallStationStatus.eRunning;
		
    eVisionStaState.eStopActive:
	     Status.StationStauts[MM_CONST.VISION_STA_HMI_STATE] := OverallStationStatus.eCycleStop;
   	
    ELSE;	
	END_CASE
END_IF
END_METHOD

METHOD PUBLIC ClearVehicleTrigger : BOOL
VAR_INPUT
END_VAR
xTrigger := FALSE;
END_METHOD

PROPERTY PUBLIC InspectionOnGoing : BOOL
GET
InspectionOnGoing := (State = eVisionStaState.eShortShotTrigger OR State = eVisionStaState.eWaitShortShotDone OR 
	                  State = eVisionStaState.eBarellInspectTrigger OR State = eVisionStaState.eWaitBarellInspectDone );
END_GET
END_PROPERTY

METHOD PUBLIC IsFaulted : BOOL
VAR_INPUT
END_VAR
IsFaulted := (State = eVisionStaState.eUnknown);
END_METHOD

PROPERTY PUBLIC Ready : BOOL
GET
Ready := (State = eVisionStaState.eReady);
END_GET
END_PROPERTY

PROPERTY PUBLIC Trigger : BOOL
SET
xTrigger := Trigger;
END_SET
END_PROPERTY

METHOD PUBLIC UpdatePartData : BOOL
VAR_INPUT

END_VAR
VAR
	TotalStainArea : DINT;
	TotalStainCount : DINT;
END_VAR
UpdatePartForHMIStatus();
PartsData.Status[VUT].VisionInspectTime := SYSTEMTIME_TO_STRING(Logging.fbCurrTime.systemTime);
IF (GVL_IO.VS_XPartEmpty) THEN
	PartsData.Status[VUT].OverallStatus := ePartStatus.eEmpty;
	RETURN;
END_IF

PartsData.Status[VUT].BurnOffTemp := GVL_IO.BU_Temperature/10; 

// Proceed down only if part is not empty
// If the Vision station is disabled then just declare that part is loaded.

IF (LotsData.Lot.VisionStationRunSelect = eVisionEnableState.Disabled) THEN   
		PartsData.Status[VUT].OverallStatus := ePartStatus.eGoodPremium;
		PartsData.Status[VUT].Premium := TRUE;	
        PartsData.Status[VUT].Good := FALSE;	
		PartsData.Status[VUT].VisionPass := TRUE;
	RETURN;
END_IF

// If only data collection then call the part loaded and collect data 
PartsData.Status[VUT].OverallStatus := ePartStatus.eLoaded; // we know its not empty from initial check

PartsData.Status[VUT].VisionData.Cam1Judgement              := GVL_IO.VS_XCam1JudgeVal;
PartsData.Status[VUT].VisionData.Cam2Judgement              := GVL_IO.VS_XCam2JudgeVal;
PartsData.Status[VUT].VisionData.Cam3Judgement              := GVL_IO.VS_XCam3JudgeVal;
PartsData.Status[VUT].VisionData.Cam4Judgement              := GVL_IO.VS_XCam4JudgeVal;

PartsData.Status[VUT].VisionData.MaxIndividualStainArea     := GVL_IO.VS_XMaxIndividualStainArea; 		
PartsData.Status[VUT].VisionData.MinIndividualStainArea	    := GVL_IO.VS_XMinIndividualStainArea; 		
PartsData.Status[VUT].VisionData.ModifiedStainArea	        := GVL_IO.VS_XModifiedStainArea;	
PartsData.Status[VUT].VisionData.ModifiedMaxStain	        := GVL_IO.VS_XModifiedMaxStain;

PartsData.Status[VUT].VisionData.XPosCam1			        := GVL_IO.VS_XXPosCam1; 		
PartsData.Status[VUT].VisionData.YPosCam1                   := GVL_IO.VS_XYPosCam1; 		
PartsData.Status[VUT].VisionData.UpperFlawAreaCam2	        := GVL_IO.VS_XUpperFlawAreaCam2;	
PartsData.Status[VUT].VisionData.LowerFlawAreaCam2	        := GVL_IO.VS_XLowerFlawAreaCam2;	
PartsData.Status[VUT].VisionData.UpperFlawCountCam2	        := GVL_IO.VS_XUpperFlawCountCam2;
PartsData.Status[VUT].VisionData.LowerFlawCountCam2	        := GVL_IO.VS_XLowerFlawCountCam2;		
PartsData.Status[VUT].VisionData.UpperFlawAreaCam3	        := GVL_IO.VS_XUpperFlawAreaCam3;	  
PartsData.Status[VUT].VisionData.LowerFlawAreaCam3	        := GVL_IO.VS_XLowerFlawAreaCam3;	
PartsData.Status[VUT].VisionData.UpperFlawCountCam3	        := GVL_IO.VS_XUpperFlawCountCam3;
PartsData.Status[VUT].VisionData.LowerFlawCountCam3	        := GVL_IO.VS_XLowerFlawCountCam3;
PartsData.Status[VUT].VisionData.UpperFlawAreaCam4	        := GVL_IO.VS_XUpperFlawAreaCam4;	 
PartsData.Status[VUT].VisionData.LowerFlawAreaCam4	        := GVL_IO.VS_XLowerFlawAreaCam4;	
PartsData.Status[VUT].VisionData.UpperFlawCountCam4	        := GVL_IO.VS_XUpperFlawCountCam4;
PartsData.Status[VUT].VisionData.LowerFlawCountCam4	        := GVL_IO.VS_XLowerFlawCountCam4;

LotsData.Lot.IndividualStainAreaMaxPremium                  := LotsData.Lot.ShortShotMinRadius;
LotsData.Lot.IndividualStainAreaMaxGood                     := LotsData.Lot.ShortShotMaxRadius;

IF (LotsData.Lot.VisionStationRunSelect = eVisionEnableState.DataCollectOnly) THEN
	  	PartsData.Status[VUT].OverallStatus := ePartStatus.eGoodPremium;
		PartsData.Status[VUT].Premium := TRUE;	
        PartsData.Status[VUT].Good := FALSE;	
		PartsData.Status[VUT].VisionPass := TRUE;
      RETURN;
END_IF

// Here on, the vision station is enabled, the part is determined to be loaded. Now check the results
IF (NOT GVL_IO.VS_XCam1JudgeVal AND NOT GVL_IO.VS_XCam2JudgeVal AND NOT GVL_IO.VS_XCam3JudgeVal AND NOT GVL_IO.VS_XCam4JudgeVal AND NOT GVL_IO.VS_XPartEmpty) THEN 
	PartsData.Status[VUT].OverallStatus := ePartStatus.eVisionPass;  // Evalute further down this method for premium or good or reject
	TotalStainArea   := (PartsData.Status[VUT].VisionData.UpperFlawAreaCam2 + PartsData.Status[VUT].VisionData.LowerFlawAreaCam2 + 
                    PartsData.Status[VUT].VisionData.UpperFlawAreaCam3 + PartsData.Status[VUT].VisionData.LowerFlawAreaCam3 + 
                    PartsData.Status[VUT].VisionData.UpperFlawAreaCam4 + PartsData.Status[VUT].VisionData.LowerFlawAreaCam4 )/1000;  
	TotalStainCount  := PartsData.Status[VUT].VisionData.UpperFlawCountCam2 + PartsData.Status[VUT].VisionData.LowerFlawCountCam2 +  					   
					PartsData.Status[VUT].VisionData.UpperFlawCountCam3 + PartsData.Status[VUT].VisionData.LowerFlawCountCam3 +    
					PartsData.Status[VUT].VisionData.UpperFlawCountCam4 + PartsData.Status[VUT].VisionData.LowerFlawCountCam4 ;   
			
	IF (PartsData.Status[VUT].VisionData.ModifiedMaxStain <= LotsData.Lot.IndividualStainAreaMaxPremium AND
        PartsData.Status[VUT].VisionData.ModifiedStainArea <= LotsData.Lot.TotalStainAreaMaxPremium AND 
        TotalStainCount <= REAL_TO_DINT(LotsData.Lot.TotalStainCountMaxPremium)) THEN
		
		PartsData.Status[VUT].OverallStatus := ePartStatus.eGoodPremium;
		PartsData.Status[VUT].Premium := TRUE;	
        PartsData.Status[VUT].Good := FALSE;	
		PartsData.Status[VUT].VisionPass := TRUE;
	ELSIF (PartsData.Status[VUT].VisionData.ModifiedMaxStain <= LotsData.Lot.IndividualStainAreaMaxGood AND
           PartsData.Status[VUT].VisionData.ModifiedStainArea <= LotsData.Lot.TotalStainAreaMaxGood AND 
           TotalStainCount <= REAL_TO_DINT(LotsData.Lot.TotalStainCountMaxGood)) THEN
		PartsData.Status[VUT].OverallStatus := ePartStatus.eGoodRegular;
        PartsData.Status[VUT].Good := TRUE;	
		PartsData.Status[VUT].Premium := FALSE;
		PartsData.Status[VUT].VisionPass := TRUE;
    ELSE 
		//PartsData.Status[VUT].OverallStatus := ePartStatus.eReject;
		PartsData.Status[VUT].OverallStatus := ePartStatus.eReject; // for now just keep calling everything as good regular, until data anlysis is complete and limits are setup
   	    PartsData.Status[VUT].Good := FALSE;
		PartsData.Status[VUT].Premium := FALSE;		
		PartsData.Status[VUT].VisionPass := FALSE;
	END_IF	 
ELSE 
	PartsData.Status[VUT].OverallStatus := ePartStatus.eReject;   
	PartsData.Status[VUT].Premium := FALSE;
    PartsData.Status[VUT].Good := FALSE;
	PartsData.Status[VUT].VisionPass := FALSE;
END_IF
END_METHOD

METHOD PUBLIC UpdatePartForHMIStatus : BOOL
VAR_INPUT
END_VAR
IF (GVL_IO.VS_XPartEmpty) THEN
	Status.VisionStatusHMI[1] := 0; // Part Empty
END_IF
Status.VisionStatusHMI[2] := BOOL_TO_INT(NOT GVL_IO.VS_XCam1JudgeVal);
Status.VisionStatusHMI[3] := DINT_TO_INT(GVL_IO.VS_XUpperFlawAreaCam2 + GVL_IO.VS_XLowerFlawAreaCam2);
Status.VisionStatusHMI[4] := DINT_TO_INT(GVL_IO.VS_XUpperFlawCountCam2 + GVL_IO.VS_XLowerFlawCountCam2);
Status.VisionStatusHMI[5] := DINT_TO_INT(GVL_IO.VS_XUpperFlawAreaCam3 + GVL_IO.VS_XLowerFlawAreaCam3);
Status.VisionStatusHMI[6] := DINT_TO_INT(GVL_IO.VS_XUpperFlawCountCam3 + GVL_IO.VS_XLowerFlawCountCam3);
Status.VisionStatusHMI[7] := DINT_TO_INT(GVL_IO.VS_XUpperFlawAreaCam4 + GVL_IO.VS_XLowerFlawAreaCam4);
Status.VisionStatusHMI[8] := DINT_TO_INT(GVL_IO.VS_XUpperFlawCountCam4 + GVL_IO.VS_XLowerFlawCountCam4);
END_METHOD

PROPERTY PUBLIC VehicleUnderTest : BYTE
GET
VehicleUnderTest := VUT;
END_GET
SET
VUT := VehicleUnderTest;
END_SET
END_PROPERTY

END_FUNCTION_BLOCK

// ---- POUs/PistonInsertStation.TcPOU
FUNCTION_BLOCK PUBLIC PistonInsertStation
VAR_INPUT
END_VAR
VAR_OUTPUT
END_VAR
VAR
	xTrigger :BOOL := FALSE; // triggers processing
	State : ePistonInsertStaState := ePistonInsertStaState.eUnknown;
	NextState : ePistonInsertStaState := ePistonInsertStaState.eUnknown;
	ErrorReturnState : ePistonInsertStaState := ePistonInsertStaState.eUnknown;
	bFirst : BOOL := TRUE;
	VUT : BYTE; //VehicleID Under Station
	DwellTimer : TON;
	StateTimer : TON;
	PartPresentTimer : TON;
END_VAR

//////////////////// ESTOP TO STATION DISABLED
// If Piston Station is disabled, then we want to make sure that we have the SMC homed and not in the way of barrels
// we also want to check if the pallet hold downs and barrel backup position are correct
// if all above conditions are true, then we want to wait in a station disabled ready state
////////////////// STATION DISABLED - STATION ENABLED
// We have to go to have a piston ready for insertion, but also have operator hit start button
/////////////////////// STATION ENABLED - STATION DISABLED
// We have to go into disabled state
//////////////////////// ESTOP- STATION ENABLED
//// Follow all the logic to get the station ready

IF (GVL_IO.MachineEStopped) THEN 
	State := ePistonInsertStaState.eUnknown;
	NextState := ePistonInsertStaState.eUnknown;
	ErrorReturnState := ePistonInsertStaState.eUnknown;
	Status.PistonStatusMsg:= 'PistonSta Unknown, Check AIR, E-STOP and Hit Start';
END_IF

CASE State OF
	
ePistonInsertStaState.eUnknown:
    Status.PistonStatusMsg:= 'PistonSta Unknown, Check AIR, E-STOP and Hit Start';
	
    GVL_IO.PI_YMtrReset := FALSE; // we need a rising edge when we do a reset
	GVL_IO.PI_YMtrSetEnable:= FALSE; // we need a rising edge when we move to the Motor Reset State in the following states
	Act_SendEscapementtoWork();
	IF (GVL_IO.MC_XStartPB AND GVL_IO.MC_XAirPressureOK  AND GVL_IO.MC_NotEStopped) THEN // wait for start button when powered up or PLC program restarted ( remove this "TRUE" after debug
		ResetDwellTimer();
		ResetStateTimer();
		LEY_MasterReset();
        NextState := ePistonInsertStaState.eSMCMtrReset;		
	END_IF	

ePistonInsertStaState.eSMCMtrReset:
    DwellTimer(IN:= TRUE, PT:= T#1S);
	IF (DwellTimer.Q) THEN
		DwellTimer(IN:=FALSE);
		GVL_IO.PI_YMtrReset := NOT GVL_IO.PI_YMtrReset; // toggle the Reset to clear Alarms
	END_IF

	IF(NOT GVL_IO.PI_XMtrAlarm) THEN
		GVL_IO.PI_YMtrReset := FALSE;
        GVL_IO.PI_YMtrSetEnable := TRUE;
		ResetDwellTimer();
		NextState := ePistonInsertStaState.eSMCMtrCheckEnabled; // change to check enabled
	END_IF
	
	StateTimer(IN:= TRUE, PT:= T#10S);
	IF (StateTimer.Q) THEN
		ErrorReturnState := ePistonInsertStaState.eSMCMtrReset;
		Status.PistonStatusMsg:= 'Unable to Reset Piston Motor, Restart LEY controller';
		ResetDwellTimer();
		ResetStateTimer();
        NextState := ePistonInsertStaState.eError;		
	END_IF
	
	

ePistonInsertStaState.eSMCMtrCheckEnabled:
   IF (GVL_IO.PI_XMtrServoEnabled AND NOT GVL_IO.PI_XMtrBusy AND NOT GVL_IO.PI_XMtrEStopped AND NOT GVL_IO.PI_XMtrAlarm) THEN
	   NextState := ePistonInsertStaState.eSMCMtrSendHome;
	   ResetDwellTimer();
   END_IF
   DwellTimer(IN:=TRUE, PT:= T#10S);
   IF (DwellTimer.Q) THEN
		ErrorReturnState := ePistonInsertStaState.eUnknown;
		Status.PistonStatusMsg:= 'Unable to Enable Piston Motor, Restart LEY controller';
		ResetDwellTimer();
		ResetStateTimer();
        NextState := ePistonInsertStaState.eError;		
	END_IF
   
 ePistonInsertStaState.eSMCMtrSendHome:
	GVL_IO.PI_YMtrGoHome := TRUE;
	IF (GVL_IO.PI_XMtrServoHomed) THEN 
		NextState := ePistonInsertStaState.eSMCMtrHomed;
		GVL_IO.PI_YMtrGoHome := FALSE;
		ResetDwellTimer();
	END_IF
	DwellTimer(IN:=TRUE, PT:= T#10S);
	IF (DwellTimer.Q) THEN
		ErrorReturnState := ePistonInsertStaState.eUnknown;
		Status.PistonStatusMsg:= 'Unable to Home Piston Motor, Clear any jams ';
		ResetDwellTimer();
		ResetStateTimer();
        NextState := ePistonInsertStaState.eError;		
	END_IF   

	   
ePistonInsertStaState.eSMCMtrHomed:
     IF (GVL_IO.PI_XMtrServoHomed AND GVL_IO.PI_XMtrServoEnabled AND NOT GVL_IO.PI_XMtrBusy (*AND GVL_IO.PI_XMtrMoveCompl*) AND GVL_IO.PI_XMtrReady) THEN
		 NextState := ePistonInsertStaState.eInit;  // not checking tool position in IMBAD2
		 ResetDwellTimer();	 
	 END_IF
	 
	DwellTimer(IN:=TRUE, PT:= T#10S);
	IF (DwellTimer.Q) THEN
		ErrorReturnState := ePistonInsertStaState.eUnknown;
		Status.PistonStatusMsg:= 'Unable to Ready Piston Motor, Restart LEY ';
		ResetDwellTimer();
		ResetStateTimer();
        NextState := ePistonInsertStaState.eError;		
	END_IF   


ePistonInsertStaState.eCheckToolPosition:
	IF (LotsData.Lot.BarrelSize = eBarrelType.Size55cc) THEN
		IF (TRUE OR GVL_IO.PI_XToolAt55_10_Barrel AND NOT GVL_IO.PI_XToolAt3_30_Barrel) THEN // no barrel backup 
			 NextState := ePistonInsertStaState.eInit;
		ELSE
			NextState := ePistonInsertStaState.eUnknown;
       		Status.PistonStatusMsg:= 'Incorrect Backup Location,Fix and Hit Start';
		END_IF
	ELSIF (LotsData.Lot.BarrelSize = eBarrelType.Size30cc) THEN
		IF (TRUE OR NOT GVL_IO.PI_XToolAt55_10_Barrel AND GVL_IO.PI_XToolAt3_30_Barrel) THEN
			 NextState := ePistonInsertStaState.eInit;
		ELSE
			NextState := ePistonInsertStaState.eUnknown;
        	Status.PistonStatusMsg:= 'Incorrect Backup Location,Fix and Hit Start';
		END_IF
	ELSE 
		NextState := ePistonInsertStaState.eUnknown;
        Status.PistonStatusMsg:= 'Incorrect Part Selection, Start New Lot';
	END_IF
	

ePistonInsertStaState.eInit:
	Act_RetractBarrelBackup();    
	Act_FreePalletHoldDown();	
	IF (GVL_IO.PI_XPistonPresentEscapement) THEN
		Act_SendEscapementtoWork();        
    ELSE 
		Act_SendEscapementToBowl();
	END_IF		
	ResetDwellTimer();
	NextState := ePistonInsertStaState.eHoming;

ePistonInsertStaState.eHoming:
    IF(IsBarrelBackupRetracted() AND IsPalletHoldDownFree()) THEN   
		ResetDwellTimer();
	 	IF (GVL_IO.PI_YEscapementToBowl) THEN // based on what direction decided in previous state
			NextState := ePistonInsertStaState.eMoveEscapemttoBowl;	
		ELSE
			NextState := ePistonInsertStaState.eMoveEscapmentToWork;
		END_IF		
	    IF (NOT LotsData.Lot.PistonInsertEnabled) THEN
			NextState := ePistonInsertStaState.eDisabledReady;
        END_IF	
	END_IF
	
	DwellTimer(IN:=TRUE, PT:= T#10S);
	IF (DwellTimer.Q) THEN
		ErrorReturnState := ePistonInsertStaState.eInit;		
		ResetDwellTimer();
		ResetStateTimer();
        NextState := ePistonInsertStaState.eError;		
	END_IF   

	
ePistonInsertStaState.eDisabledReady:
  IF (LotsData.Lot.PistonInsertEnabled) THEN
	  NextState := ePistonInsertStaState.eUnknown;
  END_IF
  IF (xTrigger) THEN
	  NextState := ePistonInsertStaState.eDepart;
  END_IF
  Status.PistonStatusMsg:= 'Station Disabled and Ready';


ePistonInsertStaState.eMoveEscapemttoBowl:
  	Act_SendEscapementToBowl();    
  	IF (IsEscapementAtBowl()) THEN
		ResetDwellTimer();
	  	NextState := ePistonInsertStaState.eEscapmentAtBowl;
  	END_IF
	
	DwellTimer(IN:=TRUE, PT:= T#10S);
	IF (DwellTimer.Q) THEN
		ErrorReturnState := ePistonInsertStaState.eMoveEscapemttoBowl;
		Status.PistonStatusMsg:= 'Escapement unable to move to Bowl,Stuck Pistons?';
		ResetDwellTimer();
		ResetStateTimer();
        NextState := ePistonInsertStaState.eError;		
	END_IF   
 
	
	 
ePistonInsertStaState.eEscapmentAtBowl:
	NextState := ePistonInsertStaState.eWaitForPartAtBowl;
	PartPresentTimer(IN:=FALSE);
	DwellTimer(IN:=FALSE);
	StateTimer(IN:=FALSE);

ePistonInsertStaState.eWaitForPartAtBowl:
    PartPresentTimer(IN:= GVL_IO.PI_XPistonPresentEscapement, PT := T#10MS); //uncommented FOR turnkey debug
	//PartPresentTimer(IN:= TRUE, PT := T#10MS); //comment this out later
    IF (PartPresentTimer.Q) THEN
		PartPresentTimer(IN:=FALSE);
		NextState := ePistonInsertStaState.eMoveEscapmentToWork;
		StateTimer(IN:=FALSE);
        ResetDwellTimer();		
	END_IF	
	
    DwellTimer(IN:=TRUE, PT:= T#10S);
	IF (DwellTimer.Q) THEN
		ErrorReturnState := ePistonInsertStaState.eMoveEscapemttoBowl;
		Status.PistonStatusMsg:= 'Piston: No Piston Detected. Is Bowl Empty? ';
		ResetDwellTimer();
		ResetStateTimer();
        NextState := ePistonInsertStaState.eError;		
	END_IF   

ePistonInsertStaState.eMoveEscapmentToWork:
 	Act_SendEscapementtoWork();
	IF (IsEscapementAtWork()) THEN
		ResetDwellTimer();
		NextState := ePistonInsertStaState.eEscapementAtWork;
	END_IF
	
	DwellTimer(IN:=TRUE, PT:= T#10S);
	IF (DwellTimer.Q) THEN
		ErrorReturnState := ePistonInsertStaState.eMoveEscapmentToWork;
		Status.PistonStatusMsg:= 'Escapement Slide Failed to go to Work';
		ResetDwellTimer();
		ResetStateTimer();
        NextState := ePistonInsertStaState.eError;		
	END_IF   


ePistonInsertStaState.eEscapementAtWork:	
	NextState := ePistonInsertStaState.eReady; // We have captured a part and now sitting on top of the motor shaft waiting for the vehicle to arrive
	

ePistonInsertStaState.eReady: // vehicle arrives to station 
	IF (xTrigger) THEN
		Act_EngagePalletHoldDown();
		Act_ExtendBarrelBackup();
		ResetDwellTimer();
        NextState := ePistonInsertStaState.ePalletHoldDownEngaged;		
		PartsData.Status[VUT].OverallStatus := ePartStatus.eReject; //define as reject upfront, later update status	          		
	END_IF
	Status.PistonStatusMsg:= 'Waiting For Vehicle To Process';

ePistonInsertStaState.ePalletHoldDownEngaged:
   Act_EngagePalletHoldDown();
   IF (IsPalletHoldDownEngaged()) THEN
	   Act_ExtendBarrelBackup();
	   ResetDwellTimer();
       NextState := ePistonInsertStaState.eWaitForBarrelBackupEngaged;   
   END_IF
   
   DwellTimer(IN:=TRUE, PT:= T#10S);
	IF (DwellTimer.Q) THEN
		ErrorReturnState := ePistonInsertStaState.ePalletHoldDownEngaged;		
		ResetDwellTimer();
		ResetStateTimer();
        NextState := ePistonInsertStaState.eError;		
	END_IF   
   
   
ePistonInsertStaState.eWaitForBarrelBackupEngaged:
	IF(IsBarrelBackupExtended()) THEN
		ResetDwellTimer();
		NextState := ePistonInsertStaState.eFirePistonUp;
	END_IF
  
	DwellTimer(IN:=TRUE, PT:= T#10S);
	IF (DwellTimer.Q) THEN
		ErrorReturnState := ePistonInsertStaState.ePalletHoldDownEngaged;		
		ResetDwellTimer();
		ResetStateTimer();
        NextState := ePistonInsertStaState.eError;		
	END_IF   

ePistonInsertStaState.eFirePistonUp:
    IF (LotsData.Lot.BarrelSize = eBarrelType.Size10cc) THEN // program 1 = 10cc
    	GVL_IO.PI_YMtrStepSelectIN0 := TRUE;
		GVL_IO.PI_YMtrStepSelectIN1 := FALSE;
	ELSIF (LotsData.Lot.BarrelSize = eBarrelType.Size5cc) THEN //program3 = 5 cc
		GVL_IO.PI_YMtrStepSelectIN0 := TRUE;
		GVL_IO.PI_YMtrStepSelectIN1 := TRUE;
	ELSE // must be 3 cc 
		GVL_IO.PI_YMtrStepSelectIN0 := FALSE; //program2 = 3cc
		GVL_IO.PI_YMtrStepSelectIN1 := TRUE;
	END_IF
	DwellTimer(IN:=TRUE,PT:= T#20MS);
	IF(DwellTimer.Q) THEN
		DwellTimer(IN:=FALSE);
		GVL_IO.PI_YMtrDriveStepTrigger:= TRUE;
		NextState := ePistonInsertStaState.eWaitForPistonStartMovUp;
	END_IF

ePistonInsertStaState.eWaitForPistonStartMovUp:
	 IF (NOT GVL_IO.PI_XMtrMoveCompl) THEN   //Piston has started to move up
		 GVL_IO.PI_YMtrDriveStepTrigger:= FALSE;
		 GVL_IO.PI_YMtrStepSelectIN0 := FALSE;
		 GVL_IO.PI_YMtrStepSelectIN1 := FALSE;
		 ResetDwellTimer();
		 NextState := ePistonInsertStaState.eWaitForPistonMovDoneUp;
	 END_IF
	DwellTimer(IN:=TRUE, PT:= T#10S);
	IF (DwellTimer.Q) THEN
		ErrorReturnState := ePistonInsertStaState.eFirePistonUp;		
		GVL_IO.PI_YMtrDriveStepTrigger:= FALSE;
		ResetDwellTimer();
		ResetStateTimer();
		Status.PistonStatusMsg:= 'SMC Mtr Possibly Jammed, Lock I/O and Home Mtr';
        NextState := ePistonInsertStaState.eError;		
	END_IF 


ePistonInsertStaState.eWaitForPistonMovDoneUp:
 	IF (GVL_IO.PI_XMtrMoveCompl) THEN
		NextState := ePistonInsertStaState.eFirePistonDown;    //There may be a way to read piston actual position
		ResetDwellTimer();
		UpdatePartData();
 	END_IF
 	DwellTimer(IN:=TRUE, PT:= T#10S);
	IF (DwellTimer.Q) THEN
		ErrorReturnState := ePistonInsertStaState.eFirePistonUp;		
		GVL_IO.PI_YMtrDriveStepTrigger:= FALSE;
		ResetDwellTimer();
		ResetStateTimer();
		Status.PistonStatusMsg:= 'SMC Mtr Possibly Jammed, Lock I/O and Home Mtr';
        NextState := ePistonInsertStaState.eError;		
	END_IF 
 

ePistonInsertStaState.eFirePistonDown:
	GVL_IO.PI_YMtrStepSelectIN0 := FALSE;
	GVL_IO.PI_YMtrStepSelectIN1 := FALSE;
	GVL_IO.PI_YMtrDriveStepTrigger:= TRUE;
	ResetDwellTimer();
	NextState := ePistonInsertStaState.eWaitForPistonStartMovDwn;

ePistonInsertStaState.eWaitForPistonStartMovDwn:
 	IF (NOT GVL_IO.PI_XMtrMoveCompl) THEN
		GVL_IO.PI_YMtrDriveStepTrigger:= FALSE;
		GVL_IO.PI_YMtrStepSelectIN0 := FALSE;
		GVL_IO.PI_YMtrStepSelectIN1 := FALSE;
		ResetDwellTimer();
	 	NextState := ePistonInsertStaState.eWaitForPistonMovDoneDown;
 	END_IF
	
	DwellTimer(IN:=TRUE, PT:= T#10S);
	IF (DwellTimer.Q) THEN
		ErrorReturnState := ePistonInsertStaState.eFirePistonDown;		
		GVL_IO.PI_YMtrDriveStepTrigger:= FALSE;
		ResetDwellTimer();
		ResetStateTimer();
		Status.PistonStatusMsg:= 'SMC Mtr Possibly Jammed, Lock I/O and Home Mtr';
        NextState := ePistonInsertStaState.eError;		
	END_IF 
  


ePistonInsertStaState.eWaitForPistonMovDoneDown:	
 	IF (GVL_IO.PI_XMtrMoveCompl) THEN
		NextState := ePistonInsertStaState.eRetractPalletHoldDownAndBarrel;
		ResetDwellTimer();
 	END_IF
	//Act_FreePalletHoldDown();   // removed at Turnkey because piston gets jammed
	//Act_RetractBarrelBackup();
	
    DwellTimer(IN:=TRUE, PT:= T#10S);
	IF (DwellTimer.Q) THEN
		ErrorReturnState := ePistonInsertStaState.eFirePistonDown;		
		GVL_IO.PI_YMtrDriveStepTrigger:= FALSE;
		ResetDwellTimer();
		ResetStateTimer();
		Status.PistonStatusMsg:= 'SMC Mtr Possibly Jammed, Lock I/O and Home Mtr';
        NextState := ePistonInsertStaState.eError;		
	END_IF 
	

 
 ePistonInsertStaState.eRetractPalletHoldDownAndBarrel:
 	Act_FreePalletHoldDown();
	Act_RetractBarrelBackup();
	ResetDwellTimer();
	NextState := ePistonInsertStaState.eWaitForPalletHoldDownAndBackupRetracted; 
 
 ePistonInsertStaState.eWaitForPalletHoldDownAndBackupRetracted:
 	IF (IsBarrelBackUpRetracted() AND IsPalletHoldDownFree()) THEN
		ResetDwellTimer();
		ResetStateTimer();
		NextState := ePistonInsertStaState.eDepart;
 	END_IF
    
